LIN {X 0,Y 129.173,Z 379.611,A -85,B 0,C 180,E1 -25427.278,E2 -25427.278} C_VEL
LIN {X 0,Y 127.042,Z 350.906,A -85,B 0,C 180,E1 -25430.039,E2 -25430.039} C_VEL
LIN {X 0,Y 126.624,Z 346.55,A -85,B 0,C 180,E1 -25430.476,E2 -25430.476} C_VEL
LIN {X 0,Y 125.446,Z 341.472,A -85,B 0,C 180,E1 -25431.146,E2 -25431.146} C_VEL
LIN {X 0,Y 123.586,Z 332.403,A -85,B 0,C 180,E1 -25437.298,E2 -25437.298} C_VEL
LIN {X 0,Y 122.03,Z 325.286,A -85,B 0,C 180,E1 -25442.561,E2 -25442.561} C_VEL
LIN {X 0,Y 121.994,Z 325.288,A -85,B 0,C 180,E1 -25449.773,E2 -25449.773} C_VEL
LIN {X 0,Y 122.194,Z 325.256,A -85,B 0,C 180,E1 -25456.694,E2 -25456.694} C_VEL
LIN {X 0,Y 122.396,Z 325.238,A -85,B 0,C 180,E1 -25460.075,E2 -25460.075} C_VEL
LIN {X 0,Y 122.56,Z 325.214,A -85,B 0,C 180,E1 -25466.706,E2 -25466.706} C_VEL
LIN {X 0,Y 123.024,Z 325.16,A -85,B 0,C 180,E1 -25469.993,E2 -25469.993} C_VEL
LIN {X 0,Y 122.41,Z 325.236,A -85,B 0,C 180,E1 -25476.586,E2 -25476.586} C_VEL
LIN {X 0,Y 122.397,Z 325.238,A -85,B 0,C 180,E1 -25479.911,E2 -25479.911} C_VEL
LIN {X 0,Y 122.188,Z 325.258,A -85,B 0,C 180,E1 -25483.293,E2 -25483.293} C_VEL
LIN {X 0,Y 121.987,Z 325.286,A -85,B 0,C 180,E1 -25490.214,E2 -25490.214} C_VEL
LIN {X 0,Y 121.947,Z 325.292,A -85,B 0,C 180,E1 -25493.782,E2 -25493.782} C_VEL
LIN {X 0,Y 121.919,Z 325.29,A -85,B 0,C 180,E1 -25500.151,E2 -25500.151} C_VEL
LIN {X 0,Y 121.87,Z 325.303,A -85,B 0,C 180,E1 -25506.159,E2 -25506.159} C_VEL
LIN {X 0,Y 121.85,Z 325.303,A -85,B 0,C 180,E1 -25511.423,E2 -25511.423} C_VEL
LIN {X 0,Y 121.846,Z 325.3,A -85,B 0,C 180,E1 -25518.559,E2 -25518.559} C_VEL
LIN {X 0,Y 121.889,Z 325.3,A -85,B 0,C 180,E1 -25524.787,E2 -25524.787} C_VEL
LIN {X 0,Y 121.907,Z 325.298,A -85,B 0,C 180,E1 -25529.832,E2 -25529.832} C_VEL
LIN {X 0,Y 121.931,Z 325.289,A -85,B 0,C 180,E1 -25536.203,E2 -25536.203} C_VEL
LIN {X 0,Y 121.964,Z 325.293,A -85,B 0,C 180,E1 -25539.771,E2 -25539.771} C_VEL
LIN {X 0,Y 122.161,Z 325.265,A -85,B 0,C 180,E1 -25546.694,E2 -25546.694} C_VEL
LIN {X 0,Y 122.367,Z 325.243,A -85,B 0,C 180,E1 -25550.077,E2 -25550.077} C_VEL
LIN {X 0,Y 122.562,Z 325.217,A -85,B 0,C 180,E1 -25556.711,E2 -25556.711} C_VEL
LIN {X 0,Y 123.006,Z 325.161,A -85,B 0,C 180,E1 -25559.998,E2 -25559.998} C_VEL
LIN {X 0,Y 122.387,Z 325.239,A -85,B 0,C 180,E1 -25566.593,E2 -25566.593} C_VEL
LIN {X 0,Y 122.367,Z 325.238,A -85,B 0,C 180,E1 -25569.92,E2 -25569.92} C_VEL
LIN {X 0,Y 122.055,Z 325.28,A -85,B 0,C 180,E1 -25576.731,E2 -25576.731} C_VEL
LIN {X 0,Y 122.002,Z 325.286,A -85,B 0,C 180,E1 -25582.856,E2 -25582.856} C_VEL
LIN {X 0,Y 121.914,Z 325.296,A -85,B 0,C 180,E1 -25587.461,E2 -25587.461} C_VEL
LIN {X 0,Y 121.874,Z 325.301,A -85,B 0,C 180,E1 -25591.263,E2 -25591.263} C_VEL
LIN {X 0,Y 121.856,Z 325.304,A -85,B 0,C 180,E1 -25596.172,E2 -25596.172} C_VEL
LIN {X 0,Y 121.899,Z 325.302,A -85,B 0,C 180,E1 -25603.44,E2 -25603.44} C_VEL
LIN {X 0,Y 123.968,Z 334.356,A -85,B 0,C 180,E1 -25609.71,E2 -25609.71} C_VEL
LIN {X 0,Y 125.965,Z 343.489,A -85,B 0,C 180,E1 -25615.496,E2 -25615.496} C_VEL
LIN {X 0,Y 129.129,Z 356.128,A -85,B 0,C 180,E1 -25616.87,E2 -25616.87} C_VEL
LIN {X 0,Y 130.258,Z 379.545,A -85,B 0,C 180,E1 -25618.925,E2 -25618.925} C_VEL
LIN {X 0,Y 130.546,Z 387.282,A -85,B 0,C 180,E1 -25619.591,E2 -25619.591} C_VEL
LIN {X 0,Y 127.713,Z 439.812,A -85,B 0,C 180,E1 -25624.001,E2 -25624.001} C_VEL
LIN {X 0,Y 127.078,Z 449.021,A -85,B 0,C 180,E1 -25625.068,E2 -25625.068} C_VEL
LIN {X 0,Y 126.116,Z 458.949,A -85,B 0,C 180,E1 -25626.616,E2 -25626.616} C_VEL
LIN {X 0,Y 125.046,Z 468.69,A -85,B 0,C 180,E1 -25628.582,E2 -25628.582} C_VEL
LIN {X 0,Y 124.012,Z 478.18,A -85,B 0,C 180,E1 -25630.991,E2 -25630.991} C_VEL
LIN {X 0,Y 122.965,Z 487.212,A -85,B 0,C 180,E1 -25633.83,E2 -25633.83} C_VEL
LIN {X 0,Y 122.171,Z 494.773,A -85,B 0,C 180,E1 -25636.705,E2 -25636.705} C_VEL
LIN {X 0,Y 121.656,Z 502.106,A -85,B 0,C 180,E1 -25640.028,E2 -25640.028} C_VEL
LIN {X 0,Y 121.435,Z 508.305,A -85,B 0,C 180,E1 -25643.361,E2 -25643.361} C_VEL
LIN {X 0,Y 121.501,Z 513.6,A -85,B 0,C 180,E1 -25646.691,E2 -25646.691} C_VEL
LIN {X 0,Y 121.483,Z 517.958,A -85,B 0,C 180,E1 -25650.007,E2 -25650.007} C_VEL
LIN {X 0,Y 121.523,Z 519.76,A -85,B 0,C 180,E1 -25651.664,E2 -25651.664} C_VEL
LIN {X 0,Y 120.888,Z 524.223,A -85,B 0,C 180,E1 -25656.683,E2 -25656.683} C_VEL
LIN {X 0,Y 120.757,Z 526.661,A -85,B 0,C 180,E1 -25660.061,E2 -25660.061} C_VEL
LIN {X 0,Y 122.013,Z 530.169,A -85,B 0,C 180,E1 -25666.744,E2 -25666.744} C_VEL
LIN {X 0,Y 125.047,Z 532.186,A -85,B 0,C 180,E1 -25673.172,E2 -25673.172} C_VEL
LIN {X 0,Y 127.347,Z 532.797,A -85,B 0,C 180,E1 -25676.204,E2 -25676.204} C_VEL
LIN {X 0,Y 132.935,Z 532.734,A -85,B 0,C 180,E1 -25681.92,E2 -25681.92} C_VEL
LIN {X 0,Y 140.05,Z 531.292,A -85,B 0,C 180,E1 -25687.029,E2 -25687.029} C_VEL
LIN {X 0,Y 144.169,Z 530.134,A -85,B 0,C 180,E1 -25689.328,E2 -25689.328} C_VEL
LIN {X 0,Y 153.238,Z 526.471,A -85,B 0,C 180,E1 -25693.47,E2 -25693.47} C_VEL
LIN {X 0,Y 160.656,Z 522.679,A -85,B 0,C 180,E1 -25696.205,E2 -25696.205} C_VEL
LIN {X 0,Y 168.584,Z 517.857,A -85,B 0,C 180,E1 -25698.625,E2 -25698.625} C_VEL
LIN {X 0,Y 176.893,Z 511.872,A -85,B 0,C 180,E1 -25700.782,E2 -25700.782} C_VEL
LIN {X 0,Y 182.966,Z 506.877,A -85,B 0,C 180,E1 -25702.125,E2 -25702.125} C_VEL
LIN {X 0,Y 186.444,Z 503.636,A -85,B 0,C 180,E1 -25702.865,E2 -25702.865} C_VEL
LIN {X 0,Y 187.553,Z 502.508,A -85,B 0,C 180,E1 -25703.38,E2 -25703.38} C_VEL
LIN {X 0,Y 187.967,Z 501.842,A -85,B 0,C 180,E1 -25704.343,E2 -25704.343} C_VEL
LIN {X 0,Y 187.307,Z 502.027,A -85,B 0,C 180,E1 -25705.711,E2 -25705.711} C_VEL
LIN {X 0,Y 185.694,Z 503.089,A -85,B 0,C 180,E1 -25707.077,E2 -25707.077} C_VEL
LIN {X 0,Y 183.227,Z 504.981,A -85,B 0,C 180,E1 -25708.567,E2 -25708.567} C_VEL
LIN {X 0,Y 179.601,Z 507.677,A -85,B 0,C 180,E1 -25710.16,E2 -25710.16} C_VEL
LIN {X 0,Y 176.658,Z 509.754,A -85,B 0,C 180,E1 -25711.01,E2 -25711.01} C_VEL
LIN {X 0,Y 169.265,Z 514.461,A -85,B 0,C 180,E1 -25712.825,E2 -25712.825} C_VEL
LIN {X 0,Y 163.188,Z 517.73,A -85,B 0,C 180,E1 -25714.491,E2 -25714.491} C_VEL
LIN {X 0,Y 154.625,Z 521.426,A -85,B 0,C 180,E1 -25717.275,E2 -25717.275} C_VEL
LIN {X 0,Y 150.902,Z 522.795,A -85,B 0,C 180,E1 -25718.665,E2 -25718.665} C_VEL
LIN {X 0,Y 141.546,Z 525.001,A -85,B 0,C 180,E1 -25722.669,E2 -25722.669} C_VEL
LIN {X 0,Y 136.899,Z 525.619,A -85,B 0,C 180,E1 -25725.128,E2 -25725.128} C_VEL
LIN {X 0,Y 132.534,Z 525.668,A -85,B 0,C 180,E1 -25727.755,E2 -25727.755} C_VEL
LIN {X 0,Y 125.02,Z 524.446,A -85,B 0,C 180,E1 -25733.546,E2 -25733.546} C_VEL
LIN {X 0,Y 121.894,Z 523.17,A -85,B 0,C 180,E1 -25736.696,E2 -25736.696} C_VEL
LIN {X 0,Y 118.039,Z 520.332,A -85,B 0,C 180,E1 -25741.708,E2 -25741.708} C_VEL
LIN {X 0,Y 115.253,Z 516.339,A -85,B 0,C 180,E1 -25747.007,E2 -25747.007} C_VEL
LIN {X 0,Y 113.524,Z 511.07,A -85,B 0,C 180,E1 -25752.516,E2 -25752.516} C_VEL
LIN {X 0,Y 112.939,Z 505.58,A -85,B 0,C 180,E1 -25757.195,E2 -25757.195} C_VEL
LIN {X 0,Y 113.016,Z 498.844,A -85,B 0,C 180,E1 -25761.91,E2 -25761.91} C_VEL
LIN {X 0,Y 113.405,Z 492.3,A -85,B 0,C 180,E1 -25765.712,E2 -25765.712} C_VEL
LIN {X 0,Y 114.052,Z 484.365,A -85,B 0,C 180,E1 -25769.538,E2 -25769.538} C_VEL
LIN {X 0,Y 114.935,Z 475.882,A -85,B 0,C 180,E1 -25772.895,E2 -25772.895} C_VEL
LIN {X 0,Y 115.837,Z 467.102,A -85,B 0,C 180,E1 -25775.732,E2 -25775.732} C_VEL
LIN {X 0,Y 117.087,Z 455.66,A -85,B 0,C 180,E1 -25778.707,E2 -25778.707} C_VEL
LIN {X 0,Y 118.276,Z 443.044,A -85,B 0,C 180,E1 -25781.1,E2 -25781.1} C_VEL
LIN {X 0,Y 118.993,Z 433.1,A -85,B 0,C 180,E1 -25782.497,E2 -25782.497} C_VEL
LIN {X 0,Y 121.054,Z 399.59,A -85,B 0,C 180,E1 -25785.835,E2 -25785.835} C_VEL
LIN {X 0,Y 122.178,Z 380.662,A -85,B 0,C 180,E1 -25787.614,E2 -25787.614} C_VEL
LIN {X 0,Y 120.099,Z 351.697,A -85,B 0,C 180,E1 -25790.566,E2 -25790.566} C_VEL
LIN {X 0,Y 119.618,Z 347.583,A -85,B 0,C 180,E1 -25791.012,E2 -25791.012} C_VEL
LIN {X 0,Y 118.244,Z 341.693,A -85,B 0,C 180,E1 -25791.746,E2 -25791.746} C_VEL
LIN {X 0,Y 116.561,Z 333.547,A -85,B 0,C 180,E1 -25797.581,E2 -25797.581} C_VEL
LIN {X 0,Y 114.949,Z 326.167,A -85,B 0,C 180,E1 -25803.315,E2 -25803.315} C_VEL
LIN {X 0,Y 114.928,Z 326.171,A -85,B 0,C 180,E1 -25808.47,E2 -25808.47} C_VEL
LIN {X 0,Y 114.972,Z 326.163,A -85,B 0,C 180,E1 -25812.198,E2 -25812.198} C_VEL
LIN {X 0,Y 115.311,Z 326.122,A -85,B 0,C 180,E1 -25819.458,E2 -25819.458} C_VEL
LIN {X 0,Y 115.487,Z 326.095,A -85,B 0,C 180,E1 -25826.504,E2 -25826.504} C_VEL
LIN {X 0,Y 115.975,Z 326.038,A -85,B 0,C 180,E1 -25829.993,E2 -25829.993} C_VEL
LIN {X 0,Y 115.352,Z 326.115,A -85,B 0,C 180,E1 -25836.991,E2 -25836.991} C_VEL
LIN {X 0,Y 115.205,Z 326.127,A -85,B 0,C 180,E1 -25842.552,E2 -25842.552} C_VEL
LIN {X 0,Y 114.966,Z 326.163,A -85,B 0,C 180,E1 -25847.788,E2 -25847.788} C_VEL
LIN {X 0,Y 114.91,Z 326.168,A -85,B 0,C 180,E1 -25853.445,E2 -25853.445} C_VEL
LIN {X 0,Y 114.847,Z 326.171,A -85,B 0,C 180,E1 -25861.046,E2 -25861.046} C_VEL
LIN {X 0,Y 114.763,Z 326.186,A -85,B 0,C 180,E1 -25867.749,E2 -25867.749} C_VEL
LIN {X 0,Y 114.764,Z 326.189,A -85,B 0,C 180,E1 -25872.702,E2 -25872.702} C_VEL
LIN {X 0,Y 114.77,Z 326.183,A -85,B 0,C 180,E1 -25877.652,E2 -25877.652} C_VEL
LIN {X 0,Y 114.765,Z 326.19,A -85,B 0,C 180,E1 -25882.739,E2 -25882.739} C_VEL
LIN {X 0,Y 114.836,Z 326.176,A -85,B 0,C 180,E1 -25888.936,E2 -25888.936} C_VEL
LIN {X 0,Y 114.894,Z 326.165,A -85,B 0,C 180,E1 -25896.538,E2 -25896.538} C_VEL
LIN {X 0,Y 114.939,Z 326.166,A -85,B 0,C 180,E1 -25902.196,E2 -25902.196} C_VEL
LIN {X 0,Y 115.281,Z 326.124,A -85,B 0,C 180,E1 -25909.46,E2 -25909.46} C_VEL
LIN {X 0,Y 115.486,Z 326.097,A -85,B 0,C 180,E1 -25916.509,E2 -25916.509} C_VEL
LIN {X 0,Y 115.958,Z 326.039,A -85,B 0,C 180,E1 -25919.998,E2 -25919.998} C_VEL
LIN {X 0,Y 115.328,Z 326.119,A -85,B 0,C 180,E1 -25926.999,E2 -25926.999} C_VEL
LIN {X 0,Y 115.179,Z 326.132,A -85,B 0,C 180,E1 -25932.56,E2 -25932.56} C_VEL
LIN {X 0,Y 114.963,Z 326.164,A -85,B 0,C 180,E1 -25937.796,E2 -25937.796} C_VEL
LIN {X 0,Y 114.92,Z 326.168,A -85,B 0,C 180,E1 -25943.492,E2 -25943.492} C_VEL
LIN {X 0,Y 114.831,Z 326.177,A -85,B 0,C 180,E1 -25951.059,E2 -25951.059} C_VEL
LIN {X 0,Y 114.751,Z 326.193,A -85,B 0,C 180,E1 -25957.765,E2 -25957.765} C_VEL
LIN {X 0,Y 114.842,Z 326.253,A -85,B 0,C 180,E1 -25962.763,E2 -25962.763} C_VEL
LIN {X 0,Y 116.972,Z 335.554,A -85,B 0,C 180,E1 -25969.512,E2 -25969.512} C_VEL
LIN {X 0,Y 118.738,Z 343.603,A -85,B 0,C 180,E1 -25974.831,E2 -25974.831} C_VEL
LIN {X 0,Y 122.146,Z 357.637,A -85,B 0,C 180,E1 -25976.43,E2 -25976.43} C_VEL
LIN {X 0,Y 123.485,Z 387.391,A -85,B 0,C 180,E1 -25979.199,E2 -25979.199} C_VEL
LIN {X 0,Y 120.627,Z 439.492,A -85,B 0,C 180,E1 -25983.868,E2 -25983.868} C_VEL
LIN {X 0,Y 119.905,Z 449.334,A -85,B 0,C 180,E1 -25985.095,E2 -25985.095} C_VEL
LIN {X 0,Y 118.97,Z 459.137,A -85,B 0,C 180,E1 -25986.741,E2 -25986.741} C_VEL
LIN {X 0,Y 117.831,Z 469.633,A -85,B 0,C 180,E1 -25989.04,E2 -25989.04} C_VEL
LIN {X 0,Y 116.793,Z 478.856,A -85,B 0,C 180,E1 -25991.593,E2 -25991.593} C_VEL
LIN {X 0,Y 115.81,Z 487.711,A -85,B 0,C 180,E1 -25994.612,E2 -25994.612} C_VEL
LIN {X 0,Y 115.05,Z 496.154,A -85,B 0,C 180,E1 -25998.123,E2 -25998.123} C_VEL
LIN {X 0,Y 114.617,Z 504.09,A -85,B 0,C 180,E1 -26002.176,E2 -26002.176} C_VEL
LIN {X 0,Y 114.643,Z 512.313,A -85,B 0,C 180,E1 -26007.372,E2 -26007.372} C_VEL
LIN {X 0,Y 114.675,Z 517.684,A -85,B 0,C 180,E1 -26011.763,E2 -26011.763} C_VEL
LIN {X 0,Y 114.045,Z 522.48,A -85,B 0,C 180,E1 -26017.086,E2 -26017.086} C_VEL
LIN {X 0,Y 114.402,Z 527.08,A -85,B 0,C 180,E1 -26024.231,E2 -26024.231} C_VEL
LIN {X 0,Y 115.32,Z 528.858,A -85,B 0,C 180,E1 -26027.747,E2 -26027.747} C_VEL
LIN {X 0,Y 118.58,Z 531.297,A -85,B 0,C 180,E1 -26034.516,E2 -26034.516} C_VEL
LIN {X 0,Y 123.784,Z 532.278,A -85,B 0,C 180,E1 -26040.734,E2 -26040.734} C_VEL
LIN {X 0,Y 128.713,Z 532.194,A -85,B 0,C 180,E1 -26045.015,E2 -26045.015} C_VEL
LIN {X 0,Y 134.453,Z 531.346,A -85,B 0,C 180,E1 -26048.851,E2 -26048.851} C_VEL
LIN {X 0,Y 143.291,Z 528.883,A -85,B 0,C 180,E1 -26053.368,E2 -26053.368} C_VEL
LIN {X 0,Y 150.718,Z 526.081,A -85,B 0,C 180,E1 -26056.285,E2 -26056.285} C_VEL
LIN {X 0,Y 158.553,Z 522.398,A -85,B 0,C 180,E1 -26058.899,E2 -26058.899} C_VEL
LIN {X 0,Y 166.866,Z 517.646,A -85,B 0,C 180,E1 -26061.186,E2 -26061.186} C_VEL
LIN {X 0,Y 175.517,Z 511.729,A -85,B 0,C 180,E1 -26063.21,E2 -26063.21} C_VEL
LIN {X 0,Y 183.776,Z 505.127,A -85,B 0,C 180,E1 -26064.843,E2 -26064.843} C_VEL
LIN {X 0,Y 190.678,Z 498.721,A -85,B 0,C 180,E1 -26066.026,E2 -26066.026} C_VEL
LIN {X 0,Y 195.373,Z 493.88,A -85,B 0,C 180,E1 -26066.764,E2 -26066.764} C_VEL
LIN {X 0,Y 195.249,Z 493.91,A -85,B 0,C 180,E1 -26067.323,E2 -26067.323} C_VEL
LIN {X 0,Y 186.903,Z 501.833,A -85,B 0,C 180,E1 -26068.868,E2 -26068.868} C_VEL
LIN {X 0,Y 179.375,Z 507.837,A -85,B 0,C 180,E1 -26070.407,E2 -26070.407} C_VEL
LIN {X 0,Y 176.658,Z 509.754,A -85,B 0,C 180,E1 -26071.01,E2 -26071.01} C_VEL
LIN {X 0,Y 172.145,Z 512.757,A -85,B 0,C 180,E1 -26071.818,E2 -26071.818} C_VEL
LIN {X 0,Y 163.776,Z 517.343,A -85,B 0,C 180,E1 -26072.782,E2 -26072.782} C_VEL
LIN {X 0,Y 155.281,Z 521.101,A -85,B 0,C 180,E1 -26073.952,E2 -26073.952} C_VEL
LIN {X 0,Y 150.639,Z 522.727,A -85,B 0,C 180,E1 -26075.114,E2 -26075.114} C_VEL
LIN {X 0,Y 144.865,Z 524.313,A -85,B 0,C 180,E1 -26077.164,E2 -26077.164} C_VEL
LIN {X 0,Y 139.439,Z 525.432,A -85,B 0,C 180,E1 -26079.342,E2 -26079.342} C_VEL
LIN {X 0,Y 132.579,Z 526.179,A -85,B 0,C 180,E1 -26082.591,E2 -26082.591} C_VEL
LIN {X 0,Y 125.145,Z 525.88,A -85,B 0,C 180,E1 -26087.02,E2 -26087.02} C_VEL
LIN {X 0,Y 121.121,Z 525.186,A -85,B 0,C 180,E1 -26089.977,E2 -26089.977} C_VEL
LIN {X 0,Y 117.53,Z 523.906,A -85,B 0,C 180,E1 -26093.133,E2 -26093.133} C_VEL
LIN {X 0,Y 111.73,Z 520.067,A -85,B 0,C 180,E1 -26100.002,E2 -26100.002} C_VEL
LIN {X 0,Y 108.67,Z 515.851,A -85,B 0,C 180,E1 -26105.569,E2 -26105.569} C_VEL
LIN {X 0,Y 107.078,Z 511.736,A -85,B 0,C 180,E1 -26110.085,E2 -26110.085} C_VEL
LIN {X 0,Y 106.121,Z 505.974,A -85,B 0,C 180,E1 -26115.363,E2 -26115.363} C_VEL
LIN {X 0,Y 105.959,Z 500.857,A -85,B 0,C 180,E1 -26119.37,E2 -26119.37} C_VEL
LIN {X 0,Y 106.315,Z 492.91,A -85,B 0,C 180,E1 -26124.406,E2 -26124.406} C_VEL
LIN {X 0,Y 106.992,Z 483.988,A -85,B 0,C 180,E1 -26128.978,E2 -26128.978} C_VEL
LIN {X 0,Y 107.971,Z 474.349,A -85,B 0,C 180,E1 -26132.979,E2 -26132.979} C_VEL
LIN {X 0,Y 109.103,Z 463.38,A -85,B 0,C 180,E1 -26136.576,E2 -26136.576} C_VEL
LIN {X 0,Y 110.273,Z 452.568,A -85,B 0,C 180,E1 -26139.3,E2 -26139.3} C_VEL
LIN {X 0,Y 111.336,Z 441.435,A -85,B 0,C 180,E1 -26141.426,E2 -26141.426} C_VEL
LIN {X 0,Y 112.092,Z 429.813,A -85,B 0,C 180,E1 -26143.045,E2 -26143.045} C_VEL
LIN {X 0,Y 115.18,Z 381.489,A -85,B 0,C 180,E1 -26147.979,E2 -26147.979} C_VEL
LIN {X 0,Y 113.117,Z 351.719,A -85,B 0,C 180,E1 -26151.205,E2 -26151.205} C_VEL
LIN {X 0,Y 111.937,Z 345.593,A -85,B 0,C 180,E1 -26151.965,E2 -26151.965} C_VEL
LIN {X 0,Y 111.009,Z 341.617,A -85,B 0,C 180,E1 -26152.595,E2 -26152.595} C_VEL
LIN {X 0,Y 109.251,Z 333.22,A -85,B 0,C 180,E1 -26159.022,E2 -26159.022} C_VEL
LIN {X 0,Y 107.849,Z 327.053,A -85,B 0,C 180,E1 -26164.14,E2 -26164.14} C_VEL
LIN {X 0,Y 107.864,Z 327.049,A -85,B 0,C 180,E1 -26170.981,E2 -26170.981} C_VEL
LIN {X 0,Y 108.211,Z 327.003,A -85,B 0,C 180,E1 -26178.758,E2 -26178.758} C_VEL
LIN {X 0,Y 108.291,Z 326.994,A -85,B 0,C 180,E1 -26182.535,E2 -26182.535} C_VEL
LIN {X 0,Y 108.901,Z 326.92,A -85,B 0,C 180,E1 -26189.993,E2 -26189.993} C_VEL
LIN {X 0,Y 108.292,Z 326.995,A -85,B 0,C 180,E1 -26197.45,E2 -26197.45} C_VEL
LIN {X 0,Y 108.139,Z 327.007,A -85,B 0,C 180,E1 -26202.866,E2 -26202.866} C_VEL
LIN {X 0,Y 107.862,Z 327.047,A -85,B 0,C 180,E1 -26209.003,E2 -26209.003} C_VEL
LIN {X 0,Y 107.825,Z 327.051,A -85,B 0,C 180,E1 -26214.14,E2 -26214.14} C_VEL
LIN {X 0,Y 107.77,Z 327.056,A -85,B 0,C 180,E1 -26222.027,E2 -26222.027} C_VEL
LIN {X 0,Y 107.671,Z 327.066,A -85,B 0,C 180,E1 -26228.435,E2 -26228.435} C_VEL
LIN {X 0,Y 107.654,Z 327.074,A -85,B 0,C 180,E1 -26235.882,E2 -26235.882} C_VEL
LIN {X 0,Y 107.665,Z 327.072,A -85,B 0,C 180,E1 -26241.546,E2 -26241.546} C_VEL
LIN {X 0,Y 107.772,Z 327.054,A -85,B 0,C 180,E1 -26248.552,E2 -26248.552} C_VEL
LIN {X 0,Y 107.858,Z 327.042,A -85,B 0,C 180,E1 -26256.984,E2 -26256.984} C_VEL
LIN {X 0,Y 107.943,Z 327.03,A -85,B 0,C 180,E1 -26264.902,E2 -26264.902} C_VEL
LIN {X 0,Y 108.199,Z 327.007,A -85,B 0,C 180,E1 -26268.761,E2 -26268.761} C_VEL
LIN {X 0,Y 108.41,Z 326.978,A -85,B 0,C 180,E1 -26276.281,E2 -26276.281} C_VEL
LIN {X 0,Y 108.884,Z 326.92,A -85,B 0,C 180,E1 -26279.998,E2 -26279.998} C_VEL
LIN {X 0,Y 108.267,Z 326.999,A -85,B 0,C 180,E1 -26287.458,E2 -26287.458} C_VEL
LIN {X 0,Y 108.113,Z 327.012,A -85,B 0,C 180,E1 -26292.874,E2 -26292.874} C_VEL
LIN {X 0,Y 107.862,Z 327.045,A -85,B 0,C 180,E1 -26299.011,E2 -26299.011} C_VEL
LIN {X 0,Y 107.83,Z 327.053,A -85,B 0,C 180,E1 -26304.182,E2 -26304.182} C_VEL
LIN {X 0,Y 107.754,Z 327.06,A -85,B 0,C 180,E1 -26312.04,E2 -26312.04} C_VEL
LIN {X 0,Y 107.671,Z 327.075,A -85,B 0,C 180,E1 -26318.458,E2 -26318.458} C_VEL
LIN {X 0,Y 107.75,Z 327.164,A -85,B 0,C 180,E1 -26321.89,E2 -26321.89} C_VEL
LIN {X 0,Y 109.811,Z 336.039,A -85,B 0,C 180,E1 -26328.762,E2 -26328.762} C_VEL
LIN {X 0,Y 111.475,Z 343.518,A -85,B 0,C 180,E1 -26334.067,E2 -26334.067} C_VEL
LIN {X 0,Y 115.169,Z 358.51,A -85,B 0,C 180,E1 -26335.917,E2 -26335.917} C_VEL
LIN {X 0,Y 116.429,Z 387.557,A -85,B 0,C 180,E1 -26338.79,E2 -26338.79} C_VEL
LIN {X 0,Y 113.507,Z 440.129,A -85,B 0,C 180,E1 -26343.833,E2 -26343.833} C_VEL
LIN {X 0,Y 112.775,Z 449.689,A -85,B 0,C 180,E1 -26345.135,E2 -26345.135} C_VEL
LIN {X 0,Y 111.816,Z 459.289,A -85,B 0,C 180,E1 -26346.88,E2 -26346.88} C_VEL
LIN {X 0,Y 110.788,Z 468.754,A -85,B 0,C 180,E1 -26349.104,E2 -26349.104} C_VEL
LIN {X 0,Y 109.939,Z 476.61,A -85,B 0,C 180,E1 -26351.369,E2 -26351.369} C_VEL
LIN {X 0,Y 108.944,Z 485.692,A -85,B 0,C 180,E1 -26354.577,E2 -26354.577} C_VEL
LIN {X 0,Y 108.164,Z 494.366,A -85,B 0,C 180,E1 -26358.338,E2 -26358.338} C_VEL
LIN {X 0,Y 107.764,Z 502.271,A -85,B 0,C 180,E1 -26362.514,E2 -26362.514} C_VEL
LIN {X 0,Y 107.771,Z 508.216,A -85,B 0,C 180,E1 -26366.269,E2 -26366.269} C_VEL
LIN {X 0,Y 107.85,Z 513.205,A -85,B 0,C 180,E1 -26370.008,E2 -26370.008} C_VEL
LIN {X 0,Y 107.724,Z 517.319,A -85,B 0,C 180,E1 -26373.748,E2 -26373.748} C_VEL
LIN {X 0,Y 107.173,Z 522.537,A -85,B 0,C 180,E1 -26380.389,E2 -26380.389} C_VEL
LIN {X 0,Y 107.702,Z 525.517,A -85,B 0,C 180,E1 -26385.137,E2 -26385.137} C_VEL
LIN {X 0,Y 110.167,Z 528.969,A -85,B 0,C 180,E1 -26392.511,E2 -26392.511} C_VEL
LIN {X 0,Y 114.837,Z 531.01,A -85,B 0,C 180,E1 -26399.319,E2 -26399.319} C_VEL
LIN {X 0,Y 117.737,Z 531.604,A -85,B 0,C 180,E1 -26402.5,E2 -26402.5} C_VEL
LIN {X 0,Y 124.879,Z 531.67,A -85,B 0,C 180,E1 -26408.251,E2 -26408.251} C_VEL
LIN {X 0,Y 133.491,Z 530.335,A -85,B 0,C 180,E1 -26413.193,E2 -26413.193} C_VEL
LIN {X 0,Y 138.224,Z 529.224,A -85,B 0,C 180,E1 -26415.387,E2 -26415.387} C_VEL
LIN {X 0,Y 148.542,Z 525.79,A -85,B 0,C 180,E1 -26419.203,E2 -26419.203} C_VEL
LIN {X 0,Y 156.816,Z 522.15,A -85,B 0,C 180,E1 -26421.657,E2 -26421.657} C_VEL
LIN {X 0,Y 165.501,Z 517.524,A -85,B 0,C 180,E1 -26423.788,E2 -26423.788} C_VEL
LIN {X 0,Y 174.882,Z 511.444,A -85,B 0,C 180,E1 -26425.716,E2 -26425.716} C_VEL
LIN {X 0,Y 180.57,Z 507.239,A -85,B 0,C 180,E1 -26426.75,E2 -26426.75} C_VEL
LIN {X 0,Y 182.251,Z 505.801,A -85,B 0,C 180,E1 -26427.326,E2 -26427.326} C_VEL
LIN {X 0,Y 171.246,Z 513.262,A -85,B 0,C 180,E1 -26429.524,E2 -26429.524} C_VEL
LIN {X 0,Y 162.55,Z 517.891,A -85,B 0,C 180,E1 -26431.603,E2 -26431.603} C_VEL
LIN {X 0,Y 156.426,Z 520.653,A -85,B 0,C 180,E1 -26433.304,E2 -26433.304} C_VEL
LIN {X 0,Y 150.639,Z 522.727,A -85,B 0,C 180,E1 -26435.114,E2 -26435.114} C_VEL
LIN {X 0,Y 147.349,Z 523.782,A -85,B 0,C 180,E1 -26435.896,E2 -26435.896} C_VEL
LIN {X 0,Y 141.039,Z 525.33,A -85,B 0,C 180,E1 -26436.675,E2 -26436.675} C_VEL
LIN {X 0,Y 134.731,Z 526.369,A -85,B 0,C 180,E1 -26437.564,E2 -26437.564} C_VEL
LIN {X 0,Y 131.496,Z 526.626,A -85,B 0,C 180,E1 -26438.551,E2 -26438.551} C_VEL
LIN {X 0,Y 122.271,Z 526.506,A -85,B 0,C 180,E1 -26443.3,E2 -26443.3} C_VEL
LIN {X 0,Y 117.777,Z 525.859,A -85,B 0,C 180,E1 -26446.193,E2 -26446.193} C_VEL
LIN {X 0,Y 110.081,Z 523.023,A -85,B 0,C 180,E1 -26452.666,E2 -26452.666} C_VEL
LIN {X 0,Y 105.478,Z 519.659,A -85,B 0,C 180,E1 -26458.164,E2 -26458.164} C_VEL
LIN {X 0,Y 102.184,Z 515.306,A -85,B 0,C 180,E1 -26463.946,E2 -26463.946} C_VEL
LIN {X 0,Y 100.176,Z 510.191,A -85,B 0,C 180,E1 -26469.576,E2 -26469.576} C_VEL
LIN {X 0,Y 99.206,Z 503.818,A -85,B 0,C 180,E1 -26475.408,E2 -26475.408} C_VEL
LIN {X 0,Y 99.173,Z 495.711,A -85,B 0,C 180,E1 -26481.499,E2 -26481.499} C_VEL
LIN {X 0,Y 99.69,Z 486.859,A -85,B 0,C 180,E1 -26486.71,E2 -26486.71} C_VEL
LIN {X 0,Y 100.37,Z 479.044,A -85,B 0,C 180,E1 -26490.453,E2 -26490.453} C_VEL
LIN {X 0,Y 101.191,Z 470.74,A -85,B 0,C 180,E1 -26493.756,E2 -26493.756} C_VEL
LIN {X 0,Y 102.221,Z 460.73,A -85,B 0,C 180,E1 -26496.986,E2 -26496.986} C_VEL
LIN {X 0,Y 103.224,Z 451.597,A -85,B 0,C 180,E1 -26499.352,E2 -26499.352} C_VEL
LIN {X 0,Y 104.235,Z 441.264,A -85,B 0,C 180,E1 -26501.446,E2 -26501.446} C_VEL
LIN {X 0,Y 105.072,Z 428.849,A -85,B 0,C 180,E1 -26503.283,E2 -26503.283} C_VEL
LIN {X 0,Y 108.147,Z 381.797,A -85,B 0,C 180,E1 -26508.447,E2 -26508.447} C_VEL
LIN {X 0,Y 105.969,Z 350.894,A -85,B 0,C 180,E1 -26512.003,E2 -26512.003} C_VEL
LIN {X 0,Y 103.793,Z 341.7,A -85,B 0,C 180,E1 -26513.359,E2 -26513.359} C_VEL
LIN {X 0,Y 102.046,Z 333.567,A -85,B 0,C 180,E1 -26520.04,E2 -26520.04} C_VEL
LIN {X 0,Y 100.808,Z 327.929,A -85,B 0,C 180,E1 -26525.007,E2 -26525.007} C_VEL
LIN {X 0,Y 100.777,Z 327.932,A -85,B 0,C 180,E1 -26529.586,E2 -26529.586} C_VEL
LIN {X 0,Y 101.121,Z 327.885,A -85,B 0,C 180,E1 -26537.958,E2 -26537.958} C_VEL
LIN {X 0,Y 101.225,Z 327.874,A -85,B 0,C 180,E1 -26542.011,E2 -26542.011} C_VEL
LIN {X 0,Y 101.828,Z 327.801,A -85,B 0,C 180,E1 -26549.992,E2 -26549.992} C_VEL
LIN {X 0,Y 101.229,Z 327.876,A -85,B 0,C 180,E1 -26557.973,E2 -26557.973} C_VEL
LIN {X 0,Y 101.051,Z 327.89,A -85,B 0,C 180,E1 -26563.164,E2 -26563.164} C_VEL
LIN {X 0,Y 100.779,Z 327.926,A -85,B 0,C 180,E1 -26570.396,E2 -26570.396} C_VEL
LIN {X 0,Y 100.73,Z 327.936,A -85,B 0,C 180,E1 -26574.898,E2 -26574.898} C_VEL
LIN {X 0,Y 100.679,Z 327.941,A -85,B 0,C 180,E1 -26583.101,E2 -26583.101} C_VEL
LIN {X 0,Y 100.622,Z 327.943,A -85,B 0,C 180,E1 -26589.795,E2 -26589.795} C_VEL
LIN {X 0,Y 100.625,Z 327.949,A -85,B 0,C 180,E1 -26595.696,E2 -26595.696} C_VEL
LIN {X 0,Y 100.604,Z 327.952,A -85,B 0,C 180,E1 -26601.041,E2 -26601.041} C_VEL
LIN {X 0,Y 100.67,Z 327.937,A -85,B 0,C 180,E1 -26606.88,E2 -26606.88} C_VEL
LIN {X 0,Y 100.714,Z 327.933,A -85,B 0,C 180,E1 -26615.084,E2 -26615.084} C_VEL
LIN {X 0,Y 100.758,Z 327.933,A -85,B 0,C 180,E1 -26619.586,E2 -26619.586} C_VEL
LIN {X 0,Y 101.098,Z 327.89,A -85,B 0,C 180,E1 -26627.96,E2 -26627.96} C_VEL
LIN {X 0,Y 101.204,Z 327.875,A -85,B 0,C 180,E1 -26632.014,E2 -26632.014} C_VEL
LIN {X 0,Y 101.812,Z 327.801,A -85,B 0,C 180,E1 -26639.998,E2 -26639.998} C_VEL
LIN {X 0,Y 101.2,Z 327.878,A -85,B 0,C 180,E1 -26647.982,E2 -26647.982} C_VEL
LIN {X 0,Y 101.047,Z 327.892,A -85,B 0,C 180,E1 -26653.223,E2 -26653.223} C_VEL
LIN {X 0,Y 100.78,Z 327.923,A -85,B 0,C 180,E1 -26660.404,E2 -26660.404} C_VEL
LIN {X 0,Y 100.752,Z 327.935,A -85,B 0,C 180,E1 -26664.962,E2 -26664.962} C_VEL
LIN {X 0,Y 100.665,Z 327.946,A -85,B 0,C 180,E1 -26673.116,E2 -26673.116} C_VEL
LIN {X 0,Y 100.68,Z 328.027,A -85,B 0,C 180,E1 -26680.92,E2 -26680.92} C_VEL
LIN {X 0,Y 102.453,Z 335.698,A -85,B 0,C 180,E1 -26687.337,E2 -26687.337} C_VEL
LIN {X 0,Y 104.234,Z 343.552,A -85,B 0,C 180,E1 -26693.296,E2 -26693.296} C_VEL
LIN {X 0,Y 108.203,Z 359.664,A -85,B 0,C 180,E1 -26695.389,E2 -26695.389} C_VEL
LIN {X 0,Y 109.373,Z 387.692,A -85,B 0,C 180,E1 -26698.344,E2 -26698.344} C_VEL
LIN {X 0,Y 106.415,Z 440.118,A -85,B 0,C 180,E1 -26703.801,E2 -26703.801} C_VEL
LIN {X 0,Y 105.687,Z 449.499,A -85,B 0,C 180,E1 -26705.191,E2 -26705.191} C_VEL
LIN {X 0,Y 104.709,Z 458.949,A -85,B 0,C 180,E1 -26707.048,E2 -26707.048} C_VEL
LIN {X 0,Y 103.805,Z 467.575,A -85,B 0,C 180,E1 -26709.19,E2 -26709.19} C_VEL
LIN {X 0,Y 102.792,Z 476.943,A -85,B 0,C 180,E1 -26712.091,E2 -26712.091} C_VEL
LIN {X 0,Y 101.856,Z 485.685,A -85,B 0,C 180,E1 -26715.44,E2 -26715.44} C_VEL
LIN {X 0,Y 101.237,Z 493.392,A -85,B 0,C 180,E1 -26719.004,E2 -26719.004} C_VEL
LIN {X 0,Y 100.903,Z 500.626,A -85,B 0,C 180,E1 -26723.008,E2 -26723.008} C_VEL
LIN {X 0,Y 100.959,Z 506.751,A -85,B 0,C 180,E1 -26727.016,E2 -26727.016} C_VEL
LIN {X 0,Y 101.154,Z 512.889,A -85,B 0,C 180,E1 -26731.999,E2 -26731.999} C_VEL
LIN {X 0,Y 100.76,Z 516.736,A -85,B 0,C 180,E1 -26736.013,E2 -26736.013} C_VEL
LIN {X 0,Y 100.727,Z 522.528,A -85,B 0,C 180,E1 -26744.142,E2 -26744.142} C_VEL
LIN {X 0,Y 102.141,Z 525.82,A -85,B 0,C 180,E1 -26750.129,E2 -26750.129} C_VEL
LIN {X 0,Y 105.977,Z 528.904,A -85,B 0,C 180,E1 -26757.665,E2 -26757.665} C_VEL
LIN {X 0,Y 108.737,Z 530.056,A -85,B 0,C 180,E1 -26761.141,E2 -26761.141} C_VEL
LIN {X 0,Y 116.682,Z 531.135,A -85,B 0,C 180,E1 -26768.465,E2 -26768.465} C_VEL
LIN {X 0,Y 123.733,Z 530.886,A -85,B 0,C 180,E1 -26772.972,E2 -26772.972} C_VEL
LIN {X 0,Y 128.42,Z 530.355,A -85,B 0,C 180,E1 -26775.356,E2 -26775.356} C_VEL
LIN {X 0,Y 138.623,Z 528.118,A -85,B 0,C 180,E1 -26779.509,E2 -26779.509} C_VEL
LIN {X 0,Y 149.665,Z 524.358,A -85,B 0,C 180,E1 -26782.968,E2 -26782.968} C_VEL
LIN {X 0,Y 158.482,Z 520.507,A -85,B 0,C 180,E1 -26785.125,E2 -26785.125} C_VEL
LIN {X 0,Y 167.573,Z 515.597,A -85,B 0,C 180,E1 -26787.014,E2 -26787.014} C_VEL
LIN {X 0,Y 165.773,Z 516.516,A -85,B 0,C 180,E1 -26787.985,E2 -26787.985} C_VEL
LIN {X 0,Y 155.932,Z 520.959,A -85,B 0,C 180,E1 -26790.28,E2 -26790.28} C_VEL
LIN {X 0,Y 146.376,Z 523.958,A -85,B 0,C 180,E1 -26793,E2 -26793} C_VEL
LIN {X 0,Y 137.879,Z 525.901,A -85,B 0,C 180,E1 -26795.936,E2 -26795.936} C_VEL
LIN {X 0,Y 131.496,Z 526.626,A -85,B 0,C 180,E1 -26798.551,E2 -26798.551} C_VEL
LIN {X 0,Y 126.981,Z 526.811,A -85,B 0,C 180,E1 -26800.248,E2 -26800.248} C_VEL
LIN {X 0,Y 122.003,Z 526.779,A -85,B 0,C 180,E1 -26801.751,E2 -26801.751} C_VEL
LIN {X 0,Y 115.298,Z 526.214,A -85,B 0,C 180,E1 -26803.788,E2 -26803.788} C_VEL
LIN {X 0,Y 109.329,Z 524.952,A -85,B 0,C 180,E1 -26806.337,E2 -26806.337} C_VEL
LIN {X 0,Y 107.002,Z 524.117,A -85,B 0,C 180,E1 -26807.95,E2 -26807.95} C_VEL
LIN {X 0,Y 100.992,Z 520.628,A -85,B 0,C 180,E1 -26814.01,E2 -26814.01} C_VEL
LIN {X 0,Y 97.821,Z 517.637,A -85,B 0,C 180,E1 -26818.398,E2 -26818.398} C_VEL
LIN {X 0,Y 94.446,Z 511.906,A -85,B 0,C 180,E1 -26825.339,E2 -26825.339} C_VEL
LIN {X 0,Y 92.805,Z 506.165,A -85,B 0,C 180,E1 -26831.25,E2 -26831.25} C_VEL
LIN {X 0,Y 92.277,Z 500.031,A -85,B 0,C 180,E1 -26836.598,E2 -26836.598} C_VEL
LIN {X 0,Y 92.329,Z 493.791,A -85,B 0,C 180,E1 -26841.199,E2 -26841.199} C_VEL
LIN {X 0,Y 92.659,Z 487.397,A -85,B 0,C 180,E1 -26845.22,E2 -26845.22} C_VEL
LIN {X 0,Y 93.351,Z 478.312,A -85,B 0,C 180,E1 -26849.921,E2 -26849.921} C_VEL
LIN {X 0,Y 94.164,Z 469.88,A -85,B 0,C 180,E1 -26853.504,E2 -26853.504} C_VEL
LIN {X 0,Y 95.009,Z 461.9,A -85,B 0,C 180,E1 -26856.286,E2 -26856.286} C_VEL
LIN {X 0,Y 96.098,Z 451.846,A -85,B 0,C 180,E1 -26859.11,E2 -26859.11} C_VEL
LIN {X 0,Y 97.186,Z 440.689,A -85,B 0,C 180,E1 -26861.517,E2 -26861.517} C_VEL
LIN {X 0,Y 98.251,Z 425.866,A -85,B 0,C 180,E1 -26863.724,E2 -26863.724} C_VEL
LIN {X 0,Y 101.016,Z 381.205,A -85,B 0,C 180,E1 -26868.966,E2 -26868.966} C_VEL
LIN {X 0,Y 98.949,Z 351.704,A -85,B 0,C 180,E1 -26872.637,E2 -26872.637} C_VEL
LIN {X 0,Y 96.574,Z 341.858,A -85,B 0,C 180,E1 -26874.148,E2 -26874.148} C_VEL
LIN {X 0,Y 95.131,Z 335.123,A -85,B 0,C 180,E1 -26880.083,E2 -26880.083} C_VEL
LIN {X 0,Y 93.705,Z 328.815,A -85,B 0,C 180,E1 -26886.072,E2 -26886.072} C_VEL
LIN {X 0,Y 93.74,Z 328.809,A -85,B 0,C 180,E1 -26892.542,E2 -26892.542} C_VEL
LIN {X 0,Y 94.022,Z 328.765,A -85,B 0,C 180,E1 -26897.034,E2 -26897.034} C_VEL
LIN {X 0,Y 94.156,Z 328.756,A -85,B 0,C 180,E1 -26901.407,E2 -26901.407} C_VEL
LIN {X 0,Y 94.758,Z 328.681,A -85,B 0,C 180,E1 -26909.991,E2 -26909.991} C_VEL
LIN {X 0,Y 94.159,Z 328.756,A -85,B 0,C 180,E1 -26918.576,E2 -26918.576} C_VEL
LIN {X 0,Y 93.959,Z 328.773,A -85,B 0,C 180,E1 -26923.488,E2 -26923.488} C_VEL
LIN {X 0,Y 93.651,Z 328.81,A -85,B 0,C 180,E1 -26932.026,E2 -26932.026} C_VEL
LIN {X 0,Y 93.595,Z 328.826,A -85,B 0,C 180,E1 -26936.765,E2 -26936.765} C_VEL
LIN {X 0,Y 93.575,Z 328.829,A -85,B 0,C 180,E1 -26944.289,E2 -26944.289} C_VEL
LIN {X 0,Y 93.514,Z 328.836,A -85,B 0,C 180,E1 -26952.545,E2 -26952.545} C_VEL
LIN {X 0,Y 93.515,Z 328.828,A -85,B 0,C 180,E1 -26958.704,E2 -26958.704} C_VEL
LIN {X 0,Y 93.566,Z 328.825,A -85,B 0,C 180,E1 -26965.69,E2 -26965.69} C_VEL
LIN {X 0,Y 93.624,Z 328.819,A -85,B 0,C 180,E1 -26974.231,E2 -26974.231} C_VEL
LIN {X 0,Y 93.632,Z 328.817,A -85,B 0,C 180,E1 -26977.955,E2 -26977.955} C_VEL
LIN {X 0,Y 93.993,Z 328.774,A -85,B 0,C 180,E1 -26987.035,E2 -26987.035} C_VEL
LIN {X 0,Y 94.134,Z 328.757,A -85,B 0,C 180,E1 -26991.41,E2 -26991.41} C_VEL
LIN {X 0,Y 94.741,Z 328.682,A -85,B 0,C 180,E1 -26999.998,E2 -26999.998} C_VEL
LIN {X 0,Y 94.129,Z 328.759,A -85,B 0,C 180,E1 -27008.586,E2 -27008.586} C_VEL
LIN {X 0,Y 93.978,Z 328.774,A -85,B 0,C 180,E1 -27013.607,E2 -27013.607} C_VEL
LIN {X 0,Y 93.662,Z 328.812,A -85,B 0,C 180,E1 -27022.033,E2 -27022.033} C_VEL
LIN {X 0,Y 93.596,Z 328.824,A -85,B 0,C 180,E1 -27026.775,E2 -27026.775} C_VEL
LIN {X 0,Y 93.563,Z 328.83,A -85,B 0,C 180,E1 -27034.307,E2 -27034.307} C_VEL
LIN {X 0,Y 93.624,Z 329.017,A -85,B 0,C 180,E1 -27039.989,E2 -27039.989} C_VEL
LIN {X 0,Y 95.548,Z 337.232,A -85,B 0,C 180,E1 -27047.35,E2 -27047.35} C_VEL
LIN {X 0,Y 96.883,Z 343.26,A -85,B 0,C 180,E1 -27052.387,E2 -27052.387} C_VEL
LIN {X 0,Y 101.24,Z 360.859,A -85,B 0,C 180,E1 -27054.879,E2 -27054.879} C_VEL
LIN {X 0,Y 102.359,Z 387.023,A -85,B 0,C 180,E1 -27057.864,E2 -27057.864} C_VEL
LIN {X 0,Y 99.381,Z 438.92,A -85,B 0,C 180,E1 -27063.64,E2 -27063.64} C_VEL
LIN {X 0,Y 98.597,Z 449.192,A -85,B 0,C 180,E1 -27065.255,E2 -27065.255} C_VEL
LIN {X 0,Y 97.622,Z 458.622,A -85,B 0,C 180,E1 -27067.246,E2 -27067.246} C_VEL
LIN {X 0,Y 96.596,Z 468.404,A -85,B 0,C 180,E1 -27069.904,E2 -27069.904} C_VEL
LIN {X 0,Y 95.619,Z 477.235,A -85,B 0,C 180,E1 -27072.913,E2 -27072.913} C_VEL
LIN {X 0,Y 94.881,Z 485.014,A -85,B 0,C 180,E1 -27076.139,E2 -27076.139} C_VEL
LIN {X 0,Y 94.28,Z 493.361,A -85,B 0,C 180,E1 -27080.354,E2 -27080.354} C_VEL
LIN {X 0,Y 94.123,Z 500.46,A -85,B 0,C 180,E1 -27084.654,E2 -27084.654} C_VEL
LIN {X 0,Y 94.314,Z 506.452,A -85,B 0,C 180,E1 -27088.941,E2 -27088.941} C_VEL
LIN {X 0,Y 94.419,Z 511.407,A -85,B 0,C 180,E1 -27093.209,E2 -27093.209} C_VEL
LIN {X 0,Y 93.93,Z 516.121,A -85,B 0,C 180,E1 -27098.614,E2 -27098.614} C_VEL
LIN {X 0,Y 94.525,Z 521.81,A -85,B 0,C 180,E1 -27107.309,E2 -27107.309} C_VEL
LIN {X 0,Y 95.696,Z 524.1,A -85,B 0,C 180,E1 -27111.55,E2 -27111.55} C_VEL
LIN {X 0,Y 99.824,Z 527.626,A -85,B 0,C 180,E1 -27119.533,E2 -27119.533} C_VEL
LIN {X 0,Y 106.119,Z 529.73,A -85,B 0,C 180,E1 -27126.593,E2 -27126.593} C_VEL
LIN {X 0,Y 110.8,Z 530.442,A -85,B 0,C 180,E1 -27130.437,E2 -27130.437} C_VEL
LIN {X 0,Y 118.65,Z 530.574,A -85,B 0,C 180,E1 -27135.304,E2 -27135.304} C_VEL
LIN {X 0,Y 128.681,Z 529.469,A -85,B 0,C 180,E1 -27139.876,E2 -27139.876} C_VEL
LIN {X 0,Y 139.722,Z 526.958,A -85,B 0,C 180,E1 -27143.593,E2 -27143.593} C_VEL
LIN {X 0,Y 148.507,Z 524.144,A -85,B 0,C 180,E1 -27145.913,E2 -27145.913} C_VEL
LIN {X 0,Y 151.519,Z 522.97,A -85,B 0,C 180,E1 -27146.607,E2 -27146.607} C_VEL
LIN {X 0,Y 153.591,Z 522.071,A -85,B 0,C 180,E1 -27147.789,E2 -27147.789} C_VEL
LIN {X 0,Y 146.865,Z 524.229,A -85,B 0,C 180,E1 -27149.471,E2 -27149.471} C_VEL
LIN {X 0,Y 136.83,Z 526.378,A -85,B 0,C 180,E1 -27152.468,E2 -27152.468} C_VEL
LIN {X 0,Y 130.922,Z 527.076,A -85,B 0,C 180,E1 -27154.569,E2 -27154.569} C_VEL
LIN {X 0,Y 120.221,Z 527.154,A -85,B 0,C 180,E1 -27159.288,E2 -27159.288} C_VEL
LIN {X 0,Y 115.01,Z 526.498,A -85,B 0,C 180,E1 -27162.211,E2 -27162.211} C_VEL
LIN {X 0,Y 107.002,Z 524.117,A -85,B 0,C 180,E1 -27167.95,E2 -27167.95} C_VEL
LIN {X 0,Y 103.558,Z 522.684,A -85,B 0,C 180,E1 -27170.433,E2 -27170.433} C_VEL
LIN {X 0,Y 96.932,Z 519.466,A -85,B 0,C 180,E1 -27174.254,E2 -27174.254} C_VEL
LIN {X 0,Y 91.012,Z 515.482,A -85,B 0,C 180,E1 -27178.471,E2 -27178.471} C_VEL
LIN {X 0,Y 88.811,Z 512.732,A -85,B 0,C 180,E1 -27181.509,E2 -27181.509} C_VEL
LIN {X 0,Y 86.525,Z 506.657,A -85,B 0,C 180,E1 -27188.175,E2 -27188.175} C_VEL
LIN {X 0,Y 85.572,Z 500.215,A -85,B 0,C 180,E1 -27194.267,E2 -27194.267} C_VEL
LIN {X 0,Y 85.437,Z 494.12,A -85,B 0,C 180,E1 -27199.213,E2 -27199.213} C_VEL
LIN {X 0,Y 85.721,Z 486.691,A -85,B 0,C 180,E1 -27204.203,E2 -27204.203} C_VEL
LIN {X 0,Y 86.275,Z 478.67,A -85,B 0,C 180,E1 -27208.676,E2 -27208.676} C_VEL
LIN {X 0,Y 87.003,Z 470.751,A -85,B 0,C 180,E1 -27212.358,E2 -27212.358} C_VEL
LIN {X 0,Y 88.006,Z 460.809,A -85,B 0,C 180,E1 -27216.118,E2 -27216.118} C_VEL
LIN {X 0,Y 89.176,Z 449.546,A -85,B 0,C 180,E1 -27219.454,E2 -27219.454} C_VEL
LIN {X 0,Y 90.479,Z 435.91,A -85,B 0,C 180,E1 -27222.348,E2 -27222.348} C_VEL
LIN {X 0,Y 92.163,Z 409.622,A -85,B 0,C 180,E1 -27225.941,E2 -27225.941} C_VEL
LIN {X 0,Y 93.939,Z 381.421,A -85,B 0,C 180,E1 -27229.459,E2 -27229.459} C_VEL
LIN {X 0,Y 91.938,Z 352.596,A -85,B 0,C 180,E1 -27233.323,E2 -27233.323} C_VEL
LIN {X 0,Y 89.386,Z 341.923,A -85,B 0,C 180,E1 -27235.069,E2 -27235.069} C_VEL
LIN {X 0,Y 87.642,Z 334.029,A -85,B 0,C 180,E1 -27242.655,E2 -27242.655} C_VEL
LIN {X 0,Y 86.645,Z 329.693,A -85,B 0,C 180,E1 -27247.331,E2 -27247.331} C_VEL
LIN {X 0,Y 86.872,Z 329.654,A -85,B 0,C 180,E1 -27256.134,E2 -27256.134} C_VEL
LIN {X 0,Y 87.062,Z 329.64,A -85,B 0,C 180,E1 -27260.7,E2 -27260.7} C_VEL
LIN {X 0,Y 87.687,Z 329.562,A -85,B 0,C 180,E1 -27269.991,E2 -27269.991} C_VEL
LIN {X 0,Y 87.062,Z 329.639,A -85,B 0,C 180,E1 -27279.281,E2 -27279.281} C_VEL
LIN {X 0,Y 86.859,Z 329.659,A -85,B 0,C 180,E1 -27284.037,E2 -27284.037} C_VEL
LIN {X 0,Y 86.597,Z 329.696,A -85,B 0,C 180,E1 -27288.931,E2 -27288.931} C_VEL
LIN {X 0,Y 86.561,Z 329.703,A -85,B 0,C 180,E1 -27296.728,E2 -27296.728} C_VEL
LIN {X 0,Y 86.492,Z 329.712,A -85,B 0,C 180,E1 -27305.649,E2 -27305.649} C_VEL
LIN {X 0,Y 86.438,Z 329.717,A -85,B 0,C 180,E1 -27312.962,E2 -27312.962} C_VEL
LIN {X 0,Y 86.437,Z 329.711,A -85,B 0,C 180,E1 -27319.42,E2 -27319.42} C_VEL
LIN {X 0,Y 86.509,Z 329.705,A -85,B 0,C 180,E1 -27325.339,E2 -27325.339} C_VEL
LIN {X 0,Y 86.547,Z 329.703,A -85,B 0,C 180,E1 -27333.252,E2 -27333.252} C_VEL
LIN {X 0,Y 86.576,Z 329.7,A -85,B 0,C 180,E1 -27341.049,E2 -27341.049} C_VEL
LIN {X 0,Y 86.838,Z 329.66,A -85,B 0,C 180,E1 -27346.151,E2 -27346.151} C_VEL
LIN {X 0,Y 87.038,Z 329.642,A -85,B 0,C 180,E1 -27350.704,E2 -27350.704} C_VEL
LIN {X 0,Y 87.671,Z 329.563,A -85,B 0,C 180,E1 -27359.998,E2 -27359.998} C_VEL
LIN {X 0,Y 87.023,Z 329.642,A -85,B 0,C 180,E1 -27369.293,E2 -27369.293} C_VEL
LIN {X 0,Y 86.87,Z 329.661,A -85,B 0,C 180,E1 -27374.044,E2 -27374.044} C_VEL
LIN {X 0,Y 86.601,Z 329.693,A -85,B 0,C 180,E1 -27378.94,E2 -27378.94} C_VEL
LIN {X 0,Y 86.56,Z 329.7,A -85,B 0,C 180,E1 -27386.765,E2 -27386.765} C_VEL
LIN {X 0,Y 86.485,Z 329.71,A -85,B 0,C 180,E1 -27395.671,E2 -27395.671} C_VEL
LIN {X 0,Y 86.541,Z 329.869,A -85,B 0,C 180,E1 -27398.819,E2 -27398.819} C_VEL
LIN {X 0,Y 88.214,Z 337.003,A -85,B 0,C 180,E1 -27405.806,E2 -27405.806} C_VEL
LIN {X 0,Y 89.625,Z 343.209,A -85,B 0,C 180,E1 -27411.467,E2 -27411.467} C_VEL
LIN {X 0,Y 94.289,Z 362.5,A -85,B 0,C 180,E1 -27414.378,E2 -27414.378} C_VEL
LIN {X 0,Y 95.275,Z 387.441,A -85,B 0,C 180,E1 -27417.436,E2 -27417.436} C_VEL
LIN {X 0,Y 92.303,Z 438.545,A -85,B 0,C 180,E1 -27423.593,E2 -27423.593} C_VEL
LIN {X 0,Y 91.516,Z 448.709,A -85,B 0,C 180,E1 -27425.331,E2 -27425.331} C_VEL
LIN {X 0,Y 90.46,Z 459.11,A -85,B 0,C 180,E1 -27427.757,E2 -27427.757} C_VEL
LIN {X 0,Y 89.37,Z 469.57,A -85,B 0,C 180,E1 -27430.949,E2 -27430.949} C_VEL
LIN {X 0,Y 88.29,Z 480.111,A -85,B 0,C 180,E1 -27435.081,E2 -27435.081} C_VEL
LIN {X 0,Y 87.482,Z 491.274,A -85,B 0,C 180,E1 -27440.764,E2 -27440.764} C_VEL
LIN {X 0,Y 87.365,Z 498.621,A -85,B 0,C 180,E1 -27445.396,E2 -27445.396} C_VEL
LIN {X 0,Y 87.714,Z 506.119,A -85,B 0,C 180,E1 -27451.157,E2 -27451.157} C_VEL
LIN {X 0,Y 87.772,Z 509.812,A -85,B 0,C 180,E1 -27454.602,E2 -27454.602} C_VEL
LIN {X 0,Y 87.251,Z 515.314,A -85,B 0,C 180,E1 -27461.626,E2 -27461.626} C_VEL
LIN {X 0,Y 88.626,Z 521.066,A -85,B 0,C 180,E1 -27470.914,E2 -27470.914} C_VEL
LIN {X 0,Y 91.264,Z 524.349,A -85,B 0,C 180,E1 -27477.526,E2 -27477.526} C_VEL
LIN {X 0,Y 96.997,Z 527.502,A -85,B 0,C 180,E1 -27485.432,E2 -27485.432} C_VEL
LIN {X 0,Y 104.576,Z 529.344,A -85,B 0,C 180,E1 -27492.231,E2 -27492.231} C_VEL
LIN {X 0,Y 109.004,Z 529.899,A -85,B 0,C 180,E1 -27495.177,E2 -27495.177} C_VEL
LIN {X 0,Y 118.898,Z 529.878,A -85,B 0,C 180,E1 -27500.217,E2 -27500.217} C_VEL
LIN {X 0,Y 129.872,Z 528.529,A -85,B 0,C 180,E1 -27504.267,E2 -27504.267} C_VEL
LIN {X 0,Y 138.029,Z 526.828,A -85,B 0,C 180,E1 -27506.633,E2 -27506.633} C_VEL
LIN {X 0,Y 140.186,Z 526.121,A -85,B 0,C 180,E1 -27507.901,E2 -27507.901} C_VEL
LIN {X 0,Y 136.349,Z 526.873,A -85,B 0,C 180,E1 -27508.975,E2 -27508.975} C_VEL
LIN {X 0,Y 127.713,Z 527.796,A -85,B 0,C 180,E1 -27511.702,E2 -27511.702} C_VEL
LIN {X 0,Y 117.983,Z 527.701,A -85,B 0,C 180,E1 -27515.553,E2 -27515.553} C_VEL
LIN {X 0,Y 112.838,Z 527.104,A -85,B 0,C 180,E1 -27518.058,E2 -27518.058} C_VEL
LIN {X 0,Y 103.111,Z 524.566,A -85,B 0,C 180,E1 -27524.181,E2 -27524.181} C_VEL
LIN {X 0,Y 97.041,Z 521.475,A -85,B 0,C 180,E1 -27529.571,E2 -27529.571} C_VEL
LIN {X 0,Y 92.104,Z 517.34,A -85,B 0,C 180,E1 -27535.626,E2 -27535.626} C_VEL
LIN {X 0,Y 88.811,Z 512.732,A -85,B 0,C 180,E1 -27541.509,E2 -27541.509} C_VEL
LIN {X 0,Y 86.972,Z 509.86,A -85,B 0,C 180,E1 -27544.586,E2 -27544.586} C_VEL
LIN {X 0,Y 84.578,Z 506.58,A -85,B 0,C 180,E1 -27547.458,E2 -27547.458} C_VEL
LIN {X 0,Y 79.455,Z 497.782,A -85,B 0,C 180,E1 -27554.171,E2 -27554.171} C_VEL
LIN {X 0,Y 78.678,Z 493.671,A -85,B 0,C 180,E1 -27557.318,E2 -27557.318} C_VEL
LIN {X 0,Y 78.864,Z 485.984,A -85,B 0,C 180,E1 -27562.95,E2 -27562.95} C_VEL
LIN {X 0,Y 79.296,Z 478.346,A -85,B 0,C 180,E1 -27567.577,E2 -27567.577} C_VEL
LIN {X 0,Y 80.01,Z 469.831,A -85,B 0,C 180,E1 -27571.808,E2 -27571.808} C_VEL
LIN {X 0,Y 80.839,Z 461.642,A -85,B 0,C 180,E1 -27575.17,E2 -27575.17} C_VEL
LIN {X 0,Y 81.979,Z 450.559,A -85,B 0,C 180,E1 -27578.794,E2 -27578.794} C_VEL
LIN {X 0,Y 83.282,Z 436.858,A -85,B 0,C 180,E1 -27582.041,E2 -27582.041} C_VEL
LIN {X 0,Y 84.87,Z 412.072,A -85,B 0,C 180,E1 -27585.796,E2 -27585.796} C_VEL
LIN {X 0,Y 86.92,Z 382.22,A -85,B 0,C 180,E1 -27589.878,E2 -27589.878} C_VEL
LIN {X 0,Y 85.081,Z 354.095,A -85,B 0,C 180,E1 -27593.938,E2 -27593.938} C_VEL
LIN {X 0,Y 82.117,Z 341.92,A -85,B 0,C 180,E1 -27596.191,E2 -27596.191} C_VEL
LIN {X 0,Y 80.441,Z 334.376,A -85,B 0,C 180,E1 -27604.089,E2 -27604.089} C_VEL
LIN {X 0,Y 79.579,Z 330.573,A -85,B 0,C 180,E1 -27608.627,E2 -27608.627} C_VEL
LIN {X 0,Y 79.795,Z 330.536,A -85,B 0,C 180,E1 -27615.669,E2 -27615.669} C_VEL
LIN {X 0,Y 79.939,Z 330.527,A -85,B 0,C 180,E1 -27619.863,E2 -27619.863} C_VEL
LIN {X 0,Y 80.617,Z 330.443,A -85,B 0,C 180,E1 -27629.99,E2 -27629.99} C_VEL
LIN {X 0,Y 79.937,Z 330.525,A -85,B 0,C 180,E1 -27640.116,E2 -27640.116} C_VEL
LIN {X 0,Y 79.687,Z 330.557,A -85,B 0,C 180,E1 -27645.33,E2 -27645.33} C_VEL
LIN {X 0,Y 79.475,Z 330.577,A -85,B 0,C 180,E1 -27650.702,E2 -27650.702} C_VEL
LIN {X 0,Y 79.462,Z 330.585,A -85,B 0,C 180,E1 -27657.81,E2 -27657.81} C_VEL
LIN {X 0,Y 79.363,Z 330.593,A -85,B 0,C 180,E1 -27662.08,E2 -27662.08} C_VEL
LIN {X 0,Y 79.352,Z 330.593,A -85,B 0,C 180,E1 -27668.297,E2 -27668.297} C_VEL
LIN {X 0,Y 79.34,Z 330.601,A -85,B 0,C 180,E1 -27675.105,E2 -27675.105} C_VEL
LIN {X 0,Y 79.367,Z 330.599,A -85,B 0,C 180,E1 -27682.816,E2 -27682.816} C_VEL
LIN {X 0,Y 79.353,Z 330.592,A -85,B 0,C 180,E1 -27687.897,E2 -27687.897} C_VEL
LIN {X 0,Y 79.488,Z 330.58,A -85,B 0,C 180,E1 -27693.76,E2 -27693.76} C_VEL
LIN {X 0,Y 79.456,Z 330.586,A -85,B 0,C 180,E1 -27699.277,E2 -27699.277} C_VEL
LIN {X 0,Y 79.764,Z 330.54,A -85,B 0,C 180,E1 -27705.681,E2 -27705.681} C_VEL
LIN {X 0,Y 79.912,Z 330.531,A -85,B 0,C 180,E1 -27709.867,E2 -27709.867} C_VEL
LIN {X 0,Y 80.601,Z 330.444,A -85,B 0,C 180,E1 -27719.997,E2 -27719.997} C_VEL
LIN {X 0,Y 79.911,Z 330.526,A -85,B 0,C 180,E1 -27730.128,E2 -27730.128} C_VEL
LIN {X 0,Y 79.703,Z 330.556,A -85,B 0,C 180,E1 -27735.336,E2 -27735.336} C_VEL
LIN {X 0,Y 79.477,Z 330.576,A -85,B 0,C 180,E1 -27740.712,E2 -27740.712} C_VEL
LIN {X 0,Y 79.457,Z 330.582,A -85,B 0,C 180,E1 -27747.843,E2 -27747.843} C_VEL
LIN {X 0,Y 79.442,Z 330.737,A -85,B 0,C 180,E1 -27757.525,E2 -27757.525} C_VEL
LIN {X 0,Y 80.863,Z 336.82,A -85,B 0,C 180,E1 -27764.047,E2 -27764.047} C_VEL
LIN {X 0,Y 82.356,Z 343.216,A -85,B 0,C 180,E1 -27770.432,E2 -27770.432} C_VEL
LIN {X 0,Y 87.304,Z 363.219,A -85,B 0,C 180,E1 -27773.748,E2 -27773.748} C_VEL
LIN {X 0,Y 88.234,Z 387.513,A -85,B 0,C 180,E1 -27776.982,E2 -27776.982} C_VEL
LIN {X 0,Y 85.224,Z 438.329,A -85,B 0,C 180,E1 -27783.702,E2 -27783.702} C_VEL
LIN {X 0,Y 84.502,Z 447.797,A -85,B 0,C 180,E1 -27785.441,E2 -27785.441} C_VEL
LIN {X 0,Y 83.468,Z 458,A -85,B 0,C 180,E1 -27787.982,E2 -27787.982} C_VEL
LIN {X 0,Y 82.533,Z 467.298,A -85,B 0,C 180,E1 -27790.972,E2 -27790.972} C_VEL
LIN {X 0,Y 81.669,Z 475.402,A -85,B 0,C 180,E1 -27794.204,E2 -27794.204} C_VEL
LIN {X 0,Y 80.938,Z 484.659,A -85,B 0,C 180,E1 -27798.745,E2 -27798.745} C_VEL
LIN {X 0,Y 80.63,Z 491.088,A -85,B 0,C 180,E1 -27802.498,E2 -27802.498} C_VEL
LIN {X 0,Y 80.708,Z 498.321,A -85,B 0,C 180,E1 -27807.515,E2 -27807.515} C_VEL
LIN {X 0,Y 81.12,Z 504.368,A -85,B 0,C 180,E1 -27812.493,E2 -27812.493} C_VEL
LIN {X 0,Y 81.177,Z 507.935,A -85,B 0,C 180,E1 -27816.222,E2 -27816.222} C_VEL
LIN {X 0,Y 80.811,Z 512.733,A -85,B 0,C 180,E1 -27822.567,E2 -27822.567} C_VEL
LIN {X 0,Y 81.714,Z 517.499,A -85,B 0,C 180,E1 -27830.131,E2 -27830.131} C_VEL
LIN {X 0,Y 84.105,Z 521.313,A -85,B 0,C 180,E1 -27837.369,E2 -27837.369} C_VEL
LIN {X 0,Y 88.032,Z 524.405,A -85,B 0,C 180,E1 -27843.983,E2 -27843.983} C_VEL
LIN {X 0,Y 91.418,Z 526.057,A -85,B 0,C 180,E1 -27847.96,E2 -27847.96} C_VEL
LIN {X 0,Y 100.517,Z 528.505,A -85,B 0,C 180,E1 -27855.641,E2 -27855.641} C_VEL
LIN {X 0,Y 109.175,Z 529.363,A -85,B 0,C 180,E1 -27860.582,E2 -27860.582} C_VEL
LIN {X 0,Y 120.037,Z 529.124,A -85,B 0,C 180,E1 -27865.056,E2 -27865.056} C_VEL
LIN {X 0,Y 125.866,Z 528.592,A -85,B 0,C 180,E1 -27866.886,E2 -27866.886} C_VEL
LIN {X 0,Y 127.11,Z 528.341,A -85,B 0,C 180,E1 -27867.986,E2 -27867.986} C_VEL
LIN {X 0,Y 117.225,Z 528.331,A -85,B 0,C 180,E1 -27871.341,E2 -27871.341} C_VEL
LIN {X 0,Y 108.44,Z 527.285,A -85,B 0,C 180,E1 -27875.145,E2 -27875.145} C_VEL
LIN {X 0,Y 100.629,Z 525.273,A -85,B 0,C 180,E1 -27879.564,E2 -27879.564} C_VEL
LIN {X 0,Y 93.679,Z 522.261,A -85,B 0,C 180,E1 -27884.82,E2 -27884.82} C_VEL
LIN {X 0,Y 87.912,Z 518.253,A -85,B 0,C 180,E1 -27890.802,E2 -27890.802} C_VEL
LIN {X 0,Y 83.551,Z 513.302,A -85,B 0,C 180,E1 -27897.351,E2 -27897.351} C_VEL
LIN {X 0,Y 80.813,Z 507.958,A -85,B 0,C 180,E1 -27903.742,E2 -27903.742} C_VEL
LIN {X 0,Y 79.182,Z 501.687,A -85,B 0,C 180,E1 -27910.228,E2 -27910.228} C_VEL
LIN {X 0,Y 78.685,Z 494.222,A -85,B 0,C 180,E1 -27916.878,E2 -27916.878} C_VEL
LIN {X 0,Y 78.678,Z 493.671,A -85,B 0,C 180,E1 -27917.318,E2 -27917.318} C_VEL
LIN {X 0,Y 78.089,Z 489.637,A -85,B 0,C 180,E1 -27920.282,E2 -27920.282} C_VEL
LIN {X 0,Y 76.749,Z 485.147,A -85,B 0,C 180,E1 -27922.958,E2 -27922.958} C_VEL
LIN {X 0,Y 73.373,Z 473.786,A -85,B 0,C 180,E1 -27928.76,E2 -27928.76} C_VEL
LIN {X 0,Y 73.076,Z 468.55,A -85,B 0,C 180,E1 -27931.25,E2 -27931.25} C_VEL
LIN {X 0,Y 74.182,Z 456.711,A -85,B 0,C 180,E1 -27936.312,E2 -27936.312} C_VEL
LIN {X 0,Y 75.322,Z 445.029,A -85,B 0,C 180,E1 -27939.906,E2 -27939.906} C_VEL
LIN {X 0,Y 76.292,Z 435.302,A -85,B 0,C 180,E1 -27942.152,E2 -27942.152} C_VEL
LIN {X 0,Y 78.72,Z 398.299,A -85,B 0,C 180,E1 -27948.036,E2 -27948.036} C_VEL
LIN {X 0,Y 79.804,Z 381.761,A -85,B 0,C 180,E1 -27950.471,E2 -27950.471} C_VEL
LIN {X 0,Y 78.077,Z 355.022,A -85,B 0,C 180,E1 -27954.696,E2 -27954.696} C_VEL
LIN {X 0,Y 74.872,Z 342.01,A -85,B 0,C 180,E1 -27957.277,E2 -27957.277} C_VEL
LIN {X 0,Y 73.207,Z 334.55,A -85,B 0,C 180,E1 -27965.911,E2 -27965.911} C_VEL
LIN {X 0,Y 72.514,Z 331.453,A -85,B 0,C 180,E1 -27969.792,E2 -27969.792} C_VEL
LIN {X 0,Y 72.831,Z 331.41,A -85,B 0,C 180,E1 -27978.862,E2 -27978.862} C_VEL
LIN {X 0,Y 73.545,Z 331.324,A -85,B 0,C 180,E1 -27989.989,E2 -27989.989} C_VEL
LIN {X 0,Y 72.828,Z 331.408,A -85,B 0,C 180,E1 -28001.116,E2 -28001.116} C_VEL
LIN {X 0,Y 72.504,Z 331.454,A -85,B 0,C 180,E1 -28006.892,E2 -28006.892} C_VEL
LIN {X 0,Y 72.364,Z 331.463,A -85,B 0,C 180,E1 -28012.845,E2 -28012.845} C_VEL
LIN {X 0,Y 72.352,Z 331.466,A -85,B 0,C 180,E1 -28019.041,E2 -28019.041} C_VEL
LIN {X 0,Y 72.281,Z 331.481,A -85,B 0,C 180,E1 -28025.671,E2 -28025.671} C_VEL
LIN {X 0,Y 72.214,Z 331.489,A -85,B 0,C 180,E1 -28032.921,E2 -28032.921} C_VEL
LIN {X 0,Y 72.274,Z 331.48,A -85,B 0,C 180,E1 -28041.046,E2 -28041.046} C_VEL
LIN {X 0,Y 72.274,Z 331.481,A -85,B 0,C 180,E1 -28044.303,E2 -28044.303} C_VEL
LIN {X 0,Y 72.342,Z 331.473,A -85,B 0,C 180,E1 -28050.935,E2 -28050.935} C_VEL
LIN {X 0,Y 72.347,Z 331.465,A -85,B 0,C 180,E1 -28057.131,E2 -28057.131} C_VEL
LIN {X 0,Y 72.657,Z 331.424,A -85,B 0,C 180,E1 -28065.239,E2 -28065.239} C_VEL
LIN {X 0,Y 72.804,Z 331.416,A -85,B 0,C 180,E1 -28068.865,E2 -28068.865} C_VEL
LIN {X 0,Y 73.528,Z 331.325,A -85,B 0,C 180,E1 -28079.997,E2 -28079.997} C_VEL
LIN {X 0,Y 72.809,Z 331.407,A -85,B 0,C 180,E1 -28091.128,E2 -28091.128} C_VEL
LIN {X 0,Y 72.54,Z 331.449,A -85,B 0,C 180,E1 -28096.894,E2 -28096.894} C_VEL
LIN {X 0,Y 72.364,Z 331.467,A -85,B 0,C 180,E1 -28102.857,E2 -28102.857} C_VEL
LIN {X 0,Y 72.338,Z 331.464,A -85,B 0,C 180,E1 -28109.06,E2 -28109.06} C_VEL
LIN {X 0,Y 72.348,Z 331.602,A -85,B 0,C 180,E1 -28116.063,E2 -28116.063} C_VEL
LIN {X 0,Y 73.868,Z 337.981,A -85,B 0,C 180,E1 -28123.609,E2 -28123.609} C_VEL
LIN {X 0,Y 75.062,Z 343.054,A -85,B 0,C 180,E1 -28129.199,E2 -28129.199} C_VEL
LIN {X 0,Y 80.346,Z 364.709,A -85,B 0,C 180,E1 -28133.214,E2 -28133.214} C_VEL
LIN {X 0,Y 81.117,Z 388.225,A -85,B 0,C 180,E1 -28136.614,E2 -28136.614} C_VEL
LIN {X 0,Y 78.139,Z 438.204,A -85,B 0,C 180,E1 -28143.849,E2 -28143.849} C_VEL
LIN {X 0,Y 77.342,Z 448.334,A -85,B 0,C 180,E1 -28145.927,E2 -28145.927} C_VEL
LIN {X 0,Y 76.293,Z 458.484,A -85,B 0,C 180,E1 -28148.762,E2 -28148.762} C_VEL
LIN {X 0,Y 75.479,Z 467.065,A -85,B 0,C 180,E1 -28151.835,E2 -28151.835} C_VEL
LIN {X 0,Y 74.55,Z 477.043,A -85,B 0,C 180,E1 -28156.381,E2 -28156.381} C_VEL
LIN {X 0,Y 73.99,Z 485.428,A -85,B 0,C 180,E1 -28161.133,E2 -28161.133} C_VEL
LIN {X 0,Y 73.932,Z 492.531,A -85,B 0,C 180,E1 -28165.923,E2 -28165.923} C_VEL
LIN {X 0,Y 74.386,Z 499.41,A -85,B 0,C 180,E1 -28171.364,E2 -28171.364} C_VEL
LIN {X 0,Y 74.713,Z 503.786,A -85,B 0,C 180,E1 -28175.408,E2 -28175.408} C_VEL
LIN {X 0,Y 74.465,Z 508.179,A -85,B 0,C 180,E1 -28180.89,E2 -28180.89} C_VEL
LIN {X 0,Y 75.456,Z 515.15,A -85,B 0,C 180,E1 -28191.883,E2 -28191.883} C_VEL
LIN {X 0,Y 79.398,Z 520.432,A -85,B 0,C 180,E1 -28202.088,E2 -28202.088} C_VEL
LIN {X 0,Y 82.419,Z 522.595,A -85,B 0,C 180,E1 -28206.656,E2 -28206.656} C_VEL
LIN {X 0,Y 90.123,Z 525.93,A -85,B 0,C 180,E1 -28214.582,E2 -28214.582} C_VEL
LIN {X 0,Y 99.588,Z 527.947,A -85,B 0,C 180,E1 -28220.927,E2 -28220.927} C_VEL
LIN {X 0,Y 110.382,Z 528.775,A -85,B 0,C 180,E1 -28225.868,E2 -28225.868} C_VEL
LIN {X 0,Y 112.409,Z 528.783,A -85,B 0,C 180,E1 -28226.624,E2 -28226.624} C_VEL
LIN {X 0,Y 114.278,Z 528.68,A -85,B 0,C 180,E1 -28228.059,E2 -28228.059} C_VEL
LIN {X 0,Y 102.798,Z 526.919,A -85,B 0,C 180,E1 -28232.726,E2 -28232.726} C_VEL
LIN {X 0,Y 98.887,Z 525.968,A -85,B 0,C 180,E1 -28234.761,E2 -28234.761} C_VEL
LIN {X 0,Y 91.261,Z 523.092,A -85,B 0,C 180,E1 -28239.616,E2 -28239.616} C_VEL
LIN {X 0,Y 84.439,Z 519.096,A -85,B 0,C 180,E1 -28245.543,E2 -28245.543} C_VEL
LIN {X 0,Y 79.09,Z 514.192,A -85,B 0,C 180,E1 -28252.239,E2 -28252.239} C_VEL
LIN {X 0,Y 75.084,Z 507.894,A -85,B 0,C 180,E1 -28260.003,E2 -28260.003} C_VEL
LIN {X 0,Y 72.961,Z 501.686,A -85,B 0,C 180,E1 -28266.919,E2 -28266.919} C_VEL
LIN {X 0,Y 72.141,Z 495.547,A -85,B 0,C 180,E1 -28273.017,E2 -28273.017} C_VEL
LIN {X 0,Y 71.979,Z 487.102,A -85,B 0,C 180,E1 -28279.986,E2 -28279.986} C_VEL
LIN {X 0,Y 72.245,Z 479.484,A -85,B 0,C 180,E1 -28285.192,E2 -28285.192} C_VEL
LIN {X 0,Y 72.816,Z 471.649,A -85,B 0,C 180,E1 -28289.685,E2 -28289.685} C_VEL
LIN {X 0,Y 73.076,Z 468.55,A -85,B 0,C 180,E1 -28291.25,E2 -28291.25} C_VEL
LIN {X 0,Y 72.806,Z 463.423,A -85,B 0,C 180,E1 -28293.517,E2 -28293.517} C_VEL
LIN {X 0,Y 70.775,Z 454.515,A -85,B 0,C 180,E1 -28296.612,E2 -28296.612} C_VEL
LIN {X 0,Y 68.839,Z 445.422,A -85,B 0,C 180,E1 -28299.339,E2 -28299.339} C_VEL
LIN {X 0,Y 68.789,Z 439.601,A -85,B 0,C 180,E1 -28300.897,E2 -28300.897} C_VEL
LIN {X 0,Y 70.109,Z 421.73,A -85,B 0,C 180,E1 -28304.443,E2 -28304.443} C_VEL
LIN {X 0,Y 72.73,Z 381.914,A -85,B 0,C 180,E1 -28311.076,E2 -28311.076} C_VEL
LIN {X 0,Y 71.072,Z 355.918,A -85,B 0,C 180,E1 -28315.554,E2 -28315.554} C_VEL
LIN {X 0,Y 67.63,Z 342.036,A -85,B 0,C 180,E1 -28318.685,E2 -28318.685} C_VEL
LIN {X 0,Y 66.232,Z 335.895,A -85,B 0,C 180,E1 -28326.541,E2 -28326.541} C_VEL
LIN {X 0,Y 65.454,Z 332.332,A -85,B 0,C 180,E1 -28331.735,E2 -28331.735} C_VEL
LIN {X 0,Y 65.726,Z 332.29,A -85,B 0,C 180,E1 -28337.64,E2 -28337.64} C_VEL
LIN {X 0,Y 66.444,Z 332.208,A -85,B 0,C 180,E1 -28349.988,E2 -28349.988} C_VEL
LIN {X 0,Y 65.721,Z 332.289,A -85,B 0,C 180,E1 -28362.336,E2 -28362.336} C_VEL
LIN {X 0,Y 65.335,Z 332.344,A -85,B 0,C 180,E1 -28368.812,E2 -28368.812} C_VEL
LIN {X 0,Y 65.213,Z 332.362,A -85,B 0,C 180,E1 -28375.52,E2 -28375.52} C_VEL
LIN {X 0,Y 65.161,Z 332.363,A -85,B 0,C 180,E1 -28382.616,E2 -28382.616} C_VEL
LIN {X 0,Y 65.157,Z 332.361,A -85,B 0,C 180,E1 -28390.966,E2 -28390.966} C_VEL
LIN {X 0,Y 65.175,Z 332.359,A -85,B 0,C 180,E1 -28399.68,E2 -28399.68} C_VEL
LIN {X 0,Y 65.208,Z 332.358,A -85,B 0,C 180,E1 -28409.533,E2 -28409.533} C_VEL
LIN {X 0,Y 65.198,Z 332.357,A -85,B 0,C 180,E1 -28414.454,E2 -28414.454} C_VEL
LIN {X 0,Y 65.56,Z 332.308,A -85,B 0,C 180,E1 -28424.684,E2 -28424.684} C_VEL
LIN {X 0,Y 65.698,Z 332.299,A -85,B 0,C 180,E1 -28427.643,E2 -28427.643} C_VEL
LIN {X 0,Y 66.427,Z 332.209,A -85,B 0,C 180,E1 -28439.997,E2 -28439.997} C_VEL
LIN {X 0,Y 65.712,Z 332.29,A -85,B 0,C 180,E1 -28452.348,E2 -28452.348} C_VEL
LIN {X 0,Y 65.349,Z 332.339,A -85,B 0,C 180,E1 -28458.819,E2 -28458.819} C_VEL
LIN {X 0,Y 65.206,Z 332.363,A -85,B 0,C 180,E1 -28465.535,E2 -28465.535} C_VEL
LIN {X 0,Y 65.176,Z 332.366,A -85,B 0,C 180,E1 -28473.544,E2 -28473.544} C_VEL
LIN {X 0,Y 65.228,Z 332.575,A -85,B 0,C 180,E1 -28474.444,E2 -28474.444} C_VEL
LIN {X 0,Y 66.58,Z 337.911,A -85,B 0,C 180,E1 -28481.569,E2 -28481.569} C_VEL
LIN {X 0,Y 67.769,Z 343.081,A -85,B 0,C 180,E1 -28487.924,E2 -28487.924} C_VEL
LIN {X 0,Y 73.218,Z 364.803,A -85,B 0,C 180,E1 -28492.361,E2 -28492.361} C_VEL
LIN {X 0,Y 74.105,Z 387.559,A -85,B 0,C 180,E1 -28495.976,E2 -28495.976} C_VEL
LIN {X 0,Y 71.031,Z 438.195,A -85,B 0,C 180,E1 -28504.151,E2 -28504.151} C_VEL
LIN {X 0,Y 70.247,Z 448.06,A -85,B 0,C 180,E1 -28506.425,E2 -28506.425} C_VEL
LIN {X 0,Y 69.35,Z 457.192,A -85,B 0,C 180,E1 -28509.24,E2 -28509.24} C_VEL
LIN {X 0,Y 68.503,Z 466.387,A -85,B 0,C 180,E1 -28512.859,E2 -28512.859} C_VEL
LIN {X 0,Y 67.751,Z 475.323,A -85,B 0,C 180,E1 -28517.279,E2 -28517.279} C_VEL
LIN {X 0,Y 67.339,Z 482.812,A -85,B 0,C 180,E1 -28521.762,E2 -28521.762} C_VEL
LIN {X 0,Y 67.304,Z 490.219,A -85,B 0,C 180,E1 -28527.02,E2 -28527.02} C_VEL
LIN {X 0,Y 67.896,Z 497.381,A -85,B 0,C 180,E1 -28532.978,E2 -28532.978} C_VEL
LIN {X 0,Y 68.323,Z 501.743,A -85,B 0,C 180,E1 -28537.399,E2 -28537.399} C_VEL
LIN {X 0,Y 68.146,Z 506.106,A -85,B 0,C 180,E1 -28543.428,E2 -28543.428} C_VEL
LIN {X 0,Y 68.804,Z 510.88,A -85,B 0,C 180,E1 -28551.075,E2 -28551.075} C_VEL
LIN {X 0,Y 71.165,Z 515.545,A -85,B 0,C 180,E1 -28559.599,E2 -28559.599} C_VEL
LIN {X 0,Y 75.336,Z 519.444,A -85,B 0,C 180,E1 -28567.337,E2 -28567.337} C_VEL
LIN {X 0,Y 80.972,Z 522.649,A -85,B 0,C 180,E1 -28573.985,E2 -28573.985} C_VEL
LIN {X 0,Y 91.907,Z 526.021,A -85,B 0,C 180,E1 -28582.287,E2 -28582.287} C_VEL
LIN {X 0,Y 100.83,Z 527.507,A -85,B 0,C 180,E1 -28586.77,E2 -28586.77} C_VEL
LIN {X 0,Y 101.777,Z 527.465,A -85,B 0,C 180,E1 -28588.128,E2 -28588.128} C_VEL
LIN {X 0,Y 97.333,Z 526.445,A -85,B 0,C 180,E1 -28590.058,E2 -28590.058} C_VEL
LIN {X 0,Y 89.336,Z 523.728,A -85,B 0,C 180,E1 -28594.365,E2 -28594.365} C_VEL
LIN {X 0,Y 81.767,Z 519.887,A -85,B 0,C 180,E1 -28599.894,E2 -28599.894} C_VEL
LIN {X 0,Y 75.362,Z 514.975,A -85,B 0,C 180,E1 -28606.521,E2 -28606.521} C_VEL
LIN {X 0,Y 70.355,Z 508.965,A -85,B 0,C 180,E1 -28614.27,E2 -28614.27} C_VEL
LIN {X 0,Y 67.47,Z 502.925,A -85,B 0,C 180,E1 -28621.495,E2 -28621.495} C_VEL
LIN {X 0,Y 65.788,Z 495.777,A -85,B 0,C 180,E1 -28629.224,E2 -28629.224} C_VEL
LIN {X 0,Y 65.295,Z 487.865,A -85,B 0,C 180,E1 -28636.659,E2 -28636.659} C_VEL
LIN {X 0,Y 65.353,Z 480.867,A -85,B 0,C 180,E1 -28642.114,E2 -28642.114} C_VEL
LIN {X 0,Y 65.791,Z 472.341,A -85,B 0,C 180,E1 -28647.626,E2 -28647.626} C_VEL
LIN {X 0,Y 66.588,Z 462.748,A -85,B 0,C 180,E1 -28652.658,E2 -28652.658} C_VEL
LIN {X 0,Y 67.652,Z 451.828,A -85,B 0,C 180,E1 -28657.148,E2 -28657.148} C_VEL
LIN {X 0,Y 68.789,Z 439.601,A -85,B 0,C 180,E1 -28660.897,E2 -28660.897} C_VEL
LIN {X 0,Y 68.647,Z 433.93,A -85,B 0,C 180,E1 -28662.239,E2 -28662.239} C_VEL
LIN {X 0,Y 66.369,Z 424.489,A -85,B 0,C 180,E1 -28663.992,E2 -28663.992} C_VEL
LIN {X 0,Y 64.015,Z 414.964,A -85,B 0,C 180,E1 -28665.618,E2 -28665.618} C_VEL
LIN {X 0,Y 63.787,Z 409.151,A -85,B 0,C 180,E1 -28666.68,E2 -28666.68} C_VEL
LIN {X 0,Y 65.649,Z 381.948,A -85,B 0,C 180,E1 -28671.655,E2 -28671.655} C_VEL
LIN {X 0,Y 64.109,Z 357.106,A -85,B 0,C 180,E1 -28676.414,E2 -28676.414} C_VEL
LIN {X 0,Y 60.371,Z 342.185,A -85,B 0,C 180,E1 -28680.094,E2 -28680.094} C_VEL
LIN {X 0,Y 59.251,Z 337.176,A -85,B 0,C 180,E1 -28687.313,E2 -28687.313} C_VEL
LIN {X 0,Y 58.484,Z 333.197,A -85,B 0,C 180,E1 -28693.528,E2 -28693.528} C_VEL
LIN {X 0,Y 58.605,Z 333.174,A -85,B 0,C 180,E1 -28696.11,E2 -28696.11} C_VEL
LIN {X 0,Y 58.773,Z 333.158,A -85,B 0,C 180,E1 -28703.119,E2 -28703.119} C_VEL
LIN {X 0,Y 59.337,Z 333.094,A -85,B 0,C 180,E1 -28709.986,E2 -28709.986} C_VEL
LIN {X 0,Y 58.773,Z 333.162,A -85,B 0,C 180,E1 -28716.853,E2 -28716.853} C_VEL
LIN {X 0,Y 58.455,Z 333.202,A -85,B 0,C 180,E1 -28725.868,E2 -28725.868} C_VEL
LIN {X 0,Y 58.155,Z 333.231,A -85,B 0,C 180,E1 -28731.239,E2 -28731.239} C_VEL
LIN {X 0,Y 58.12,Z 333.238,A -85,B 0,C 180,E1 -28738.908,E2 -28738.908} C_VEL
LIN {X 0,Y 58.006,Z 333.255,A -85,B 0,C 180,E1 -28747.264,E2 -28747.264} C_VEL
LIN {X 0,Y 57.986,Z 333.255,A -85,B 0,C 180,E1 -28756.627,E2 -28756.627} C_VEL
LIN {X 0,Y 58.001,Z 333.261,A -85,B 0,C 180,E1 -28762.705,E2 -28762.705} C_VEL
LIN {X 0,Y 58.109,Z 333.246,A -85,B 0,C 180,E1 -28771.063,E2 -28771.063} C_VEL
LIN {X 0,Y 58.138,Z 333.239,A -85,B 0,C 180,E1 -28778.733,E2 -28778.733} C_VEL
LIN {X 0,Y 58.571,Z 333.18,A -85,B 0,C 180,E1 -28786.111,E2 -28786.111} C_VEL
LIN {X 0,Y 58.754,Z 333.157,A -85,B 0,C 180,E1 -28793.126,E2 -28793.126} C_VEL
LIN {X 0,Y 59.32,Z 333.094,A -85,B 0,C 180,E1 -28799.996,E2 -28799.996} C_VEL
LIN {X 0,Y 58.756,Z 333.166,A -85,B 0,C 180,E1 -28806.866,E2 -28806.866} C_VEL
LIN {X 0,Y 58.48,Z 333.201,A -85,B 0,C 180,E1 -28816.036,E2 -28816.036} C_VEL
LIN {X 0,Y 58.122,Z 333.235,A -85,B 0,C 180,E1 -28828.921,E2 -28828.921} C_VEL
LIN {X 0,Y 58.165,Z 333.277,A -85,B 0,C 180,E1 -28832.278,E2 -28832.278} C_VEL
LIN {X 0,Y 59.521,Z 338.779,A -85,B 0,C 180,E1 -28840.493,E2 -28840.493} C_VEL
LIN {X 0,Y 60.542,Z 343.19,A -85,B 0,C 180,E1 -28846.475,E2 -28846.475} C_VEL
LIN {X 0,Y 66.075,Z 365.178,A -85,B 0,C 180,E1 -28851.525,E2 -28851.525} C_VEL
LIN {X 0,Y 66.432,Z 371.61,A -85,B 0,C 180,E1 -28852.69,E2 -28852.69} C_VEL
LIN {X 0,Y 67.008,Z 387.877,A -85,B 0,C 180,E1 -28855.554,E2 -28855.554} C_VEL
LIN {X 0,Y 63.948,Z 438.062,A -85,B 0,C 180,E1 -28864.593,E2 -28864.593} C_VEL
LIN {X 0,Y 63.175,Z 447.77,A -85,B 0,C 180,E1 -28867.101,E2 -28867.101} C_VEL
LIN {X 0,Y 62.319,Z 456.875,A -85,B 0,C 180,E1 -28870.241,E2 -28870.241} C_VEL
LIN {X 0,Y 61.558,Z 466.052,A -85,B 0,C 180,E1 -28874.282,E2 -28874.282} C_VEL
LIN {X 0,Y 60.907,Z 474.935,A -85,B 0,C 180,E1 -28879.207,E2 -28879.207} C_VEL
LIN {X 0,Y 60.637,Z 482.339,A -85,B 0,C 180,E1 -28884.193,E2 -28884.193} C_VEL
LIN {X 0,Y 60.901,Z 489.666,A -85,B 0,C 180,E1 -28890.013,E2 -28890.013} C_VEL
LIN {X 0,Y 61.786,Z 496.693,A -85,B 0,C 180,E1 -28896.544,E2 -28896.544} C_VEL
LIN {X 0,Y 62.114,Z 499.497,A -85,B 0,C 180,E1 -28899.784,E2 -28899.784} C_VEL
LIN {X 0,Y 62.01,Z 504.019,A -85,B 0,C 180,E1 -28906.472,E2 -28906.472} C_VEL
LIN {X 0,Y 63.489,Z 509.735,A -85,B 0,C 180,E1 -28916.293,E2 -28916.293} C_VEL
LIN {X 0,Y 68.408,Z 515.8,A -85,B 0,C 180,E1 -28928.066,E2 -28928.066} C_VEL
LIN {X 0,Y 74.066,Z 519.514,A -85,B 0,C 180,E1 -28935.38,E2 -28935.38} C_VEL
LIN {X 0,Y 80.906,Z 522.479,A -85,B 0,C 180,E1 -28941.434,E2 -28941.434} C_VEL
LIN {X 0,Y 88.329,Z 524.72,A -85,B 0,C 180,E1 -28946.157,E2 -28946.157} C_VEL
LIN {X 0,Y 89.862,Z 524.88,A -85,B 0,C 180,E1 -28948.139,E2 -28948.139} C_VEL
LIN {X 0,Y 79.963,Z 520.585,A -85,B 0,C 180,E1 -28953.934,E2 -28953.934} C_VEL
LIN {X 0,Y 72.545,Z 515.801,A -85,B 0,C 180,E1 -28960.183,E2 -28960.183} C_VEL
LIN {X 0,Y 66.523,Z 509.88,A -85,B 0,C 180,E1 -28967.805,E2 -28967.805} C_VEL
LIN {X 0,Y 62.074,Z 502.746,A -85,B 0,C 180,E1 -28976.758,E2 -28976.758} C_VEL
LIN {X 0,Y 59.768,Z 495.597,A -85,B 0,C 180,E1 -28985.063,E2 -28985.063} C_VEL
LIN {X 0,Y 58.9,Z 488.905,A -85,B 0,C 180,E1 -28992.056,E2 -28992.056} C_VEL
LIN {X 0,Y 58.673,Z 481.392,A -85,B 0,C 180,E1 -28998.802,E2 -28998.802} C_VEL
LIN {X 0,Y 58.907,Z 472.111,A -85,B 0,C 180,E1 -29005.63,E2 -29005.63} C_VEL
LIN {X 0,Y 59.606,Z 462.379,A -85,B 0,C 180,E1 -29011.332,E2 -29011.332} C_VEL
LIN {X 0,Y 60.511,Z 452.159,A -85,B 0,C 180,E1 -29016.018,E2 -29016.018} C_VEL
LIN {X 0,Y 61.697,Z 439.439,A -85,B 0,C 180,E1 -29020.386,E2 -29020.386} C_VEL
LIN {X 0,Y 63.08,Z 420.226,A -85,B 0,C 180,E1 -29024.557,E2 -29024.557} C_VEL
LIN {X 0,Y 63.787,Z 409.151,A -85,B 0,C 180,E1 -29026.68,E2 -29026.68} C_VEL
LIN {X 0,Y 63.682,Z 403.382,A -85,B 0,C 180,E1 -29027.78,E2 -29027.78} C_VEL
LIN {X 0,Y 61.693,Z 393.925,A -85,B 0,C 180,E1 -29029.691,E2 -29029.691} C_VEL
LIN {X 0,Y 58.822,Z 382.566,A -85,B 0,C 180,E1 -29032.19,E2 -29032.19} C_VEL
LIN {X 0,Y 58.321,Z 378.7,A -85,B 0,C 180,E1 -29033.034,E2 -29033.034} C_VEL
LIN {X 0,Y 57.31,Z 358.891,A -85,B 0,C 180,E1 -29037.28,E2 -29037.28} C_VEL
LIN {X 0,Y 53.149,Z 342.366,A -85,B 0,C 180,E1 -29041.881,E2 -29041.881} C_VEL
LIN {X 0,Y 51.849,Z 336.456,A -85,B 0,C 180,E1 -29051.604,E2 -29051.604} C_VEL
LIN {X 0,Y 51.565,Z 334.051,A -85,B 0,C 180,E1 -29056.186,E2 -29056.186} C_VEL
LIN {X 0,Y 52.223,Z 333.98,A -85,B 0,C 180,E1 -29069.984,E2 -29069.984} C_VEL
LIN {X 0,Y 51.649,Z 334.051,A -85,B 0,C 180,E1 -29077.804,E2 -29077.804} C_VEL
LIN {X 0,Y 51.335,Z 334.09,A -85,B 0,C 180,E1 -29086.584,E2 -29086.584} C_VEL
LIN {X 0,Y 50.994,Z 334.129,A -85,B 0,C 180,E1 -29094.402,E2 -29094.402} C_VEL
LIN {X 0,Y 51,Z 334.132,A -85,B 0,C 180,E1 -29104.219,E2 -29104.219} C_VEL
LIN {X 0,Y 50.953,Z 334.132,A -85,B 0,C 180,E1 -29116.391,E2 -29116.391} C_VEL
LIN {X 0,Y 50.994,Z 334.123,A -85,B 0,C 180,E1 -29126.54,E2 -29126.54} C_VEL
LIN {X 0,Y 50.98,Z 334.124,A -85,B 0,C 180,E1 -29135.566,E2 -29135.566} C_VEL
LIN {X 0,Y 51.354,Z 334.078,A -85,B 0,C 180,E1 -29144.111,E2 -29144.111} C_VEL
LIN {X 0,Y 51.629,Z 334.047,A -85,B 0,C 180,E1 -29152.172,E2 -29152.172} C_VEL
LIN {X 0,Y 52.206,Z 333.979,A -85,B 0,C 180,E1 -29159.996,E2 -29159.996} C_VEL
LIN {X 0,Y 51.634,Z 334.053,A -85,B 0,C 180,E1 -29167.819,E2 -29167.819} C_VEL
LIN {X 0,Y 51.339,Z 334.09,A -85,B 0,C 180,E1 -29176.689,E2 -29176.689} C_VEL
LIN {X 0,Y 51.142,Z 334.221,A -85,B 0,C 180,E1 -29189.873,E2 -29189.873} C_VEL
LIN {X 0,Y 52.49,Z 339.899,A -85,B 0,C 180,E1 -29199.722,E2 -29199.722} C_VEL
LIN {X 0,Y 53.197,Z 343.037,A -85,B 0,C 180,E1 -29204.57,E2 -29204.57} C_VEL
LIN {X 0,Y 57.539,Z 359.63,A -85,B 0,C 180,E1 -29209.088,E2 -29209.088} C_VEL
LIN {X 0,Y 59.353,Z 368.408,A -85,B 0,C 180,E1 -29211.151,E2 -29211.151} C_VEL
LIN {X 0,Y 59.96,Z 387.747,A -85,B 0,C 180,E1 -29214.968,E2 -29214.968} C_VEL
LIN {X 0,Y 56.838,Z 438.723,A -85,B 0,C 180,E1 -29225.353,E2 -29225.353} C_VEL
LIN {X 0,Y 56.016,Z 448.635,A -85,B 0,C 180,E1 -29228.392,E2 -29228.392} C_VEL
LIN {X 0,Y 55.199,Z 458.383,A -85,B 0,C 180,E1 -29232.416,E2 -29232.416} C_VEL
LIN {X 0,Y 54.463,Z 468.6,A -85,B 0,C 180,E1 -29237.912,E2 -29237.912} C_VEL
LIN {X 0,Y 54.125,Z 479.399,A -85,B 0,C 180,E1 -29245.361,E2 -29245.361} C_VEL
LIN {X 0,Y 54.737,Z 488.976,A -85,B 0,C 180,E1 -29253.695,E2 -29253.695} C_VEL
LIN {X 0,Y 55.864,Z 495.907,A -85,B 0,C 180,E1 -29260.891,E2 -29260.891} C_VEL
LIN {X 0,Y 55.955,Z 499.584,A -85,B 0,C 180,E1 -29266.429,E2 -29266.429} C_VEL
LIN {X 0,Y 57.814,Z 506.716,A -85,B 0,C 180,E1 -29279.107,E2 -29279.107} C_VEL
LIN {X 0,Y 63.306,Z 513.31,A -85,B 0,C 180,E1 -29291.779,E2 -29291.779} C_VEL
LIN {X 0,Y 71.834,Z 518.406,A -85,B 0,C 180,E1 -29301.519,E2 -29301.519} C_VEL
LIN {X 0,Y 76.834,Z 520.5,A -85,B 0,C 180,E1 -29305.42,E2 -29305.42} C_VEL
LIN {X 0,Y 79.05,Z 521.231,A -85,B 0,C 180,E1 -29307.765,E2 -29307.765} C_VEL
LIN {X 0,Y 70.695,Z 516.462,A -85,B 0,C 180,E1 -29313.486,E2 -29313.486} C_VEL
LIN {X 0,Y 62.547,Z 509.636,A -85,B 0,C 180,E1 -29322.005,E2 -29322.005} C_VEL
LIN {X 0,Y 57.767,Z 503.423,A -85,B 0,C 180,E1 -29329.894,E2 -29329.894} C_VEL
LIN {X 0,Y 54.62,Z 496.832,A -85,B 0,C 180,E1 -29338.161,E2 -29338.161} C_VEL
LIN {X 0,Y 52.748,Z 488.679,A -85,B 0,C 180,E1 -29347.661,E2 -29347.661} C_VEL
LIN {X 0,Y 52.164,Z 480.664,A -85,B 0,C 180,E1 -29355.636,E2 -29355.636} C_VEL
LIN {X 0,Y 52.159,Z 472.214,A -85,B 0,C 180,E1 -29362.637,E2 -29362.637} C_VEL
LIN {X 0,Y 52.613,Z 462.855,A -85,B 0,C 180,E1 -29368.966,E2 -29368.966} C_VEL
LIN {X 0,Y 53.355,Z 452.912,A -85,B 0,C 180,E1 -29374.291,E2 -29374.291} C_VEL
LIN {X 0,Y 54.144,Z 444.185,A -85,B 0,C 180,E1 -29377.955,E2 -29377.955} C_VEL
LIN {X 0,Y 55.151,Z 433.186,A -85,B 0,C 180,E1 -29381.385,E2 -29381.385} C_VEL
LIN {X 0,Y 58.624,Z 383.822,A -85,B 0,C 180,E1 -29391.95,E2 -29391.95} C_VEL
LIN {X 0,Y 58.321,Z 378.7,A -85,B 0,C 180,E1 -29393.034,E2 -29393.034} C_VEL
LIN {X 0,Y 57.295,Z 373.005,A -85,B 0,C 180,E1 -29394.349,E2 -29394.349} C_VEL
LIN {X 0,Y 53.864,Z 363.995,A -85,B 0,C 180,E1 -29396.863,E2 -29396.863} C_VEL
LIN {X 0,Y 50.587,Z 356.919,A -85,B 0,C 180,E1 -29399.149,E2 -29399.149} C_VEL
LIN {X 0,Y 47.9,Z 349.636,A -85,B 0,C 180,E1 -29401.62,E2 -29401.62} C_VEL
LIN {X 0,Y 45.878,Z 342.2,A -85,B 0,C 180,E1 -29404.437,E2 -29404.437} C_VEL
LIN {X 0,Y 44.76,Z 336.137,A -85,B 0,C 180,E1 -29416.369,E2 -29416.369} C_VEL
LIN {X 0,Y 44.499,Z 334.939,A -85,B 0,C 180,E1 -29419.176,E2 -29419.176} C_VEL
LIN {X 0,Y 45.1,Z 334.867,A -85,B 0,C 180,E1 -29429.982,E2 -29429.982} C_VEL
LIN {X 0,Y 44.494,Z 334.942,A -85,B 0,C 180,E1 -29439.069,E2 -29439.069} C_VEL
LIN {X 0,Y 44.103,Z 334.989,A -85,B 0,C 180,E1 -29448.563,E2 -29448.563} C_VEL
LIN {X 0,Y 43.806,Z 335.02,A -85,B 0,C 180,E1 -29458.746,E2 -29458.746} C_VEL
LIN {X 0,Y 43.817,Z 335.023,A -85,B 0,C 180,E1 -29466.672,E2 -29466.672} C_VEL
LIN {X 0,Y 43.765,Z 335.025,A -85,B 0,C 180,E1 -29480.027,E2 -29480.027} C_VEL
LIN {X 0,Y 43.795,Z 335.029,A -85,B 0,C 180,E1 -29491.216,E2 -29491.216} C_VEL
LIN {X 0,Y 44.162,Z 334.978,A -85,B 0,C 180,E1 -29502.634,E2 -29502.634} C_VEL
LIN {X 0,Y 44.47,Z 334.943,A -85,B 0,C 180,E1 -29510.902,E2 -29510.902} C_VEL
LIN {X 0,Y 45.082,Z 334.866,A -85,B 0,C 180,E1 -29519.995,E2 -29519.995} C_VEL
LIN {X 0,Y 44.494,Z 334.938,A -85,B 0,C 180,E1 -29529.083,E2 -29529.083} C_VEL
LIN {X 0,Y 44.119,Z 334.982,A -85,B 0,C 180,E1 -29538.573,E2 -29538.573} C_VEL
LIN {X 0,Y 43.99,Z 335.108,A -85,B 0,C 180,E1 -29546.696,E2 -29546.696} C_VEL
LIN {X 0,Y 45.086,Z 339.532,A -85,B 0,C 180,E1 -29555.765,E2 -29555.765} C_VEL
LIN {X 0,Y 45.894,Z 342.917,A -85,B 0,C 180,E1 -29562.194,E2 -29562.194} C_VEL
LIN {X 0,Y 50.334,Z 359.705,A -85,B 0,C 180,E1 -29567.642,E2 -29567.642} C_VEL
LIN {X 0,Y 52.351,Z 369.081,A -85,B 0,C 180,E1 -29570.157,E2 -29570.157} C_VEL
LIN {X 0,Y 52.852,Z 388.408,A -85,B 0,C 180,E1 -29574.497,E2 -29574.497} C_VEL
LIN {X 0,Y 49.854,Z 437.738,A -85,B 0,C 180,E1 -29586.111,E2 -29586.111} C_VEL
LIN {X 0,Y 49.059,Z 447.735,A -85,B 0,C 180,E1 -29589.582,E2 -29589.582} C_VEL
LIN {X 0,Y 48.335,Z 457.582,A -85,B 0,C 180,E1 -29594.198,E2 -29594.198} C_VEL
LIN {X 0,Y 47.753,Z 467.825,A -85,B 0,C 180,E1 -29600.488,E2 -29600.488} C_VEL
LIN {X 0,Y 47.698,Z 478.611,A -85,B 0,C 180,E1 -29608.962,E2 -29608.962} C_VEL
LIN {X 0,Y 48.792,Z 488.237,A -85,B 0,C 180,E1 -29618.298,E2 -29618.298} C_VEL
LIN {X 0,Y 49.968,Z 493.389,A -85,B 0,C 180,E1 -29624.264,E2 -29624.264} C_VEL
LIN {X 0,Y 50.683,Z 499.334,A -85,B 0,C 180,E1 -29634.597,E2 -29634.597} C_VEL
LIN {X 0,Y 54.228,Z 506.268,A -85,B 0,C 180,E1 -29647.922,E2 -29647.922} C_VEL
LIN {X 0,Y 62.963,Z 513.406,A -85,B 0,C 180,E1 -29661.398,E2 -29661.398} C_VEL
LIN {X 0,Y 67.872,Z 516.027,A -85,B 0,C 180,E1 -29665.946,E2 -29665.946} C_VEL
LIN {X 0,Y 68.267,Z 516.064,A -85,B 0,C 180,E1 -29667.608,E2 -29667.608} C_VEL
LIN {X 0,Y 59.307,Z 509.23,A -85,B 0,C 180,E1 -29675.5,E2 -29675.5} C_VEL
LIN {X 0,Y 53.873,Z 503.349,A -85,B 0,C 180,E1 -29682.935,E2 -29682.935} C_VEL
LIN {X 0,Y 49.704,Z 496.405,A -85,B 0,C 180,E1 -29691.876,E2 -29691.876} C_VEL
LIN {X 0,Y 47.041,Z 488.252,A -85,B 0,C 180,E1 -29702.145,E2 -29702.145} C_VEL
LIN {X 0,Y 45.925,Z 480.42,A -85,B 0,C 180,E1 -29711.033,E2 -29711.033} C_VEL
LIN {X 0,Y 45.562,Z 473.211,A -85,B 0,C 180,E1 -29717.974,E2 -29717.974} C_VEL
LIN {X 0,Y 45.677,Z 464.656,A -85,B 0,C 180,E1 -29724.848,E2 -29724.848} C_VEL
LIN {X 0,Y 46.222,Z 455.413,A -85,B 0,C 180,E1 -29730.88,E2 -29730.88} C_VEL
LIN {X 0,Y 47.053,Z 445.263,A -85,B 0,C 180,E1 -29736.029,E2 -29736.029} C_VEL
LIN {X 0,Y 47.965,Z 434.412,A -85,B 0,C 180,E1 -29740.075,E2 -29740.075} C_VEL
LIN {X 0,Y 50.46,Z 396.323,A -85,B 0,C 180,E1 -29749.812,E2 -29749.812} C_VEL
LIN {X 0,Y 51.529,Z 382.319,A -85,B 0,C 180,E1 -29753.055,E2 -29753.055} C_VEL
LIN {X 0,Y 50.226,Z 359.39,A -85,B 0,C 180,E1 -29758.631,E2 -29758.631} C_VEL
LIN {X 0,Y 47.9,Z 349.636,A -85,B 0,C 180,E1 -29761.62,E2 -29761.62} C_VEL
LIN {X 0,Y 46.305,Z 346.285,A -85,B 0,C 180,E1 -29763.303,E2 -29763.303} C_VEL
LIN {X 0,Y 44.026,Z 343.609,A -85,B 0,C 180,E1 -29765.79,E2 -29765.79} C_VEL
LIN {X 0,Y 40.795,Z 340.785,A -85,B 0,C 180,E1 -29770.425,E2 -29770.425} C_VEL
LIN {X 0,Y 38.31,Z 338.259,A -85,B 0,C 180,E1 -29776.648,E2 -29776.648} C_VEL
LIN {X 0,Y 37.715,Z 336.928,A -85,B 0,C 180,E1 -29780.203,E2 -29780.203} C_VEL
LIN {X 0,Y 37.537,Z 335.8,A -85,B 0,C 180,E1 -29783.259,E2 -29783.259} C_VEL
LIN {X 0,Y 37.959,Z 335.756,A -85,B 0,C 180,E1 -29789.979,E2 -29789.979} C_VEL
LIN {X 0,Y 37.274,Z 335.834,A -85,B 0,C 180,E1 -29800.845,E2 -29800.845} C_VEL
LIN {X 0,Y 37.026,Z 335.87,A -85,B 0,C 180,E1 -29808.35,E2 -29808.35} C_VEL
LIN {X 0,Y 36.697,Z 335.914,A -85,B 0,C 180,E1 -29825.037,E2 -29825.037} C_VEL
LIN {X 0,Y 36.701,Z 335.902,A -85,B 0,C 180,E1 -29829.997,E2 -29829.997} C_VEL
LIN {X 0,Y 36.691,Z 335.905,A -85,B 0,C 180,E1 -29839.971,E2 -29839.971} C_VEL
LIN {X 0,Y 36.678,Z 335.909,A -85,B 0,C 180,E1 -29844.904,E2 -29844.904} C_VEL
LIN {X 0,Y 37.011,Z 335.872,A -85,B 0,C 180,E1 -29861.615,E2 -29861.615} C_VEL
LIN {X 0,Y 37.269,Z 335.843,A -85,B 0,C 180,E1 -29869.124,E2 -29869.124} C_VEL
LIN {X 0,Y 37.94,Z 335.754,A -85,B 0,C 180,E1 -29879.994,E2 -29879.994} C_VEL
LIN {X 0,Y 37.294,Z 335.829,A -85,B 0,C 180,E1 -29890.856,E2 -29890.856} C_VEL
LIN {X 0,Y 36.957,Z 336.012,A -85,B 0,C 180,E1 -29902.348,E2 -29902.348} C_VEL
LIN {X 0,Y 38.021,Z 340.453,A -85,B 0,C 180,E1 -29913.672,E2 -29913.672} C_VEL
LIN {X 0,Y 38.644,Z 342.854,A -85,B 0,C 180,E1 -29919.106,E2 -29919.106} C_VEL
LIN {X 0,Y 42.546,Z 357.386,A -85,B 0,C 180,E1 -29925.001,E2 -29925.001} C_VEL
LIN {X 0,Y 45.323,Z 369.95,A -85,B 0,C 180,E1 -29929.1,E2 -29929.1} C_VEL
LIN {X 0,Y 45.753,Z 388.434,A -85,B 0,C 180,E1 -29933.916,E2 -29933.916} C_VEL
LIN {X 0,Y 42.837,Z 437.556,A -85,B 0,C 180,E1 -29947.409,E2 -29947.409} C_VEL
LIN {X 0,Y 42.137,Z 446.838,A -85,B 0,C 180,E1 -29951.169,E2 -29951.169} C_VEL
LIN {X 0,Y 41.522,Z 456.761,A -85,B 0,C 180,E1 -29956.564,E2 -29956.564} C_VEL
LIN {X 0,Y 41.183,Z 465.458,A -85,B 0,C 180,E1 -29962.667,E2 -29962.667} C_VEL
LIN {X 0,Y 41.361,Z 473.958,A -85,B 0,C 180,E1 -29970.02,E2 -29970.02} C_VEL
LIN {X 0,Y 42.26,Z 482.132,A -85,B 0,C 180,E1 -29978.386,E2 -29978.386} C_VEL
LIN {X 0,Y 43.993,Z 489.324,A -85,B 0,C 180,E1 -29986.661,E2 -29986.661} C_VEL
LIN {X 0,Y 44.521,Z 492.03,A -85,B 0,C 180,E1 -29990.822,E2 -29990.822} C_VEL
LIN {X 0,Y 47.253,Z 500.098,A -85,B 0,C 180,E1 -30006.524,E2 -30006.524} C_VEL
LIN {X 0,Y 54.364,Z 507.465,A -85,B 0,C 180,E1 -30020.882,E2 -30020.882} C_VEL
LIN {X 0,Y 59.123,Z 510.592,A -85,B 0,C 180,E1 -30026.331,E2 -30026.331} C_VEL
LIN {X 0,Y 51.842,Z 504.094,A -85,B 0,C 180,E1 -30033.863,E2 -30033.863} C_VEL
LIN {X 0,Y 46.43,Z 497.377,A -85,B 0,C 180,E1 -30042.383,E2 -30042.383} C_VEL
LIN {X 0,Y 42.553,Z 489.85,A -85,B 0,C 180,E1 -30052.384,E2 -30052.384} C_VEL
LIN {X 0,Y 40.453,Z 482.047,A -85,B 0,C 180,E1 -30062.495,E2 -30062.495} C_VEL
LIN {X 0,Y 39.418,Z 474.127,A -85,B 0,C 180,E1 -30071.576,E2 -30071.576} C_VEL
LIN {X 0,Y 39.096,Z 464.199,A -85,B 0,C 180,E1 -30081.077,E2 -30081.077} C_VEL
LIN {X 0,Y 39.393,Z 455.293,A -85,B 0,C 180,E1 -30087.972,E2 -30087.972} C_VEL
LIN {X 0,Y 40.058,Z 445.155,A -85,B 0,C 180,E1 -30094.009,E2 -30094.009} C_VEL
LIN {X 0,Y 40.952,Z 434.009,A -85,B 0,C 180,E1 -30098.871,E2 -30098.871} C_VEL
LIN {X 0,Y 43.371,Z 396.618,A -85,B 0,C 180,E1 -30110.029,E2 -30110.029} C_VEL
LIN {X 0,Y 44.443,Z 382.324,A -85,B 0,C 180,E1 -30113.863,E2 -30113.863} C_VEL
LIN {X 0,Y 43.273,Z 360.437,A -85,B 0,C 180,E1 -30120.087,E2 -30120.087} C_VEL
LIN {X 0,Y 39.7,Z 345.977,A -85,B 0,C 180,E1 -30125.659,E2 -30125.659} C_VEL
LIN {X 0,Y 38.556,Z 342.199,A -85,B 0,C 180,E1 -30127.731,E2 -30127.731} C_VEL
LIN {X 0,Y 37.799,Z 337.288,A -85,B 0,C 180,E1 -30139.264,E2 -30139.264} C_VEL
LIN {X 0,Y 37.715,Z 336.928,A -85,B 0,C 180,E1 -30140.203,E2 -30140.203} C_VEL
LIN {X 0,Y 36.876,Z 336.061,A -85,B 0,C 180,E1 -30144.573,E2 -30144.573} C_VEL
LIN {X 0,Y 34.838,Z 336.14,A -85,B 0,C 180,E1 -30151.067,E2 -30151.067} C_VEL
LIN {X 0,Y 29.543,Z 336.66,A -85,B 0,C 180,E1 -30174.471,E2 -30174.471} C_VEL
LIN {X 0,Y 29.468,Z 336.675,A -85,B 0,C 180,E1 -30178.455,E2 -30178.455} C_VEL
LIN {X 0,Y 29.521,Z 336.67,A -85,B 0,C 180,E1 -30195.533,E2 -30195.533} C_VEL
LIN {X 0,Y 29.452,Z 336.678,A -85,B 0,C 180,E1 -30211.486,E2 -30211.486} C_VEL
LIN {X 0,Y 29.821,Z 336.643,A -85,B 0,C 180,E1 -30220.41,E2 -30220.41} C_VEL
LIN {X 0,Y 30.055,Z 336.619,A -85,B 0,C 180,E1 -30226.47,E2 -30226.47} C_VEL
LIN {X 0,Y 30.757,Z 336.555,A -85,B 0,C 180,E1 -30239.993,E2 -30239.993} C_VEL
LIN {X 0,Y 30.022,Z 336.731,A -85,B 0,C 180,E1 -30255.451,E2 -30255.451} C_VEL
LIN {X 0,Y 30.994,Z 341.443,A -85,B 0,C 180,E1 -30270.669,E2 -30270.669} C_VEL
LIN {X 0,Y 31.3,Z 342.811,A -85,B 0,C 180,E1 -30274.628,E2 -30274.628} C_VEL
LIN {X 0,Y 34.309,Z 353.117,A -85,B 0,C 180,E1 -30280.437,E2 -30280.437} C_VEL
LIN {X 0,Y 38.205,Z 369.895,A -85,B 0,C 180,E1 -30287.369,E2 -30287.369} C_VEL
LIN {X 0,Y 38.671,Z 388.642,A -85,B 0,C 180,E1 -30293.188,E2 -30293.188} C_VEL
LIN {X 0,Y 35.869,Z 437.018,A -85,B 0,C 180,E1 -30309.225,E2 -30309.225} C_VEL
LIN {X 0,Y 35.271,Z 446.867,A -85,B 0,C 180,E1 -30314.124,E2 -30314.124} C_VEL
LIN {X 0,Y 34.891,Z 455.585,A -85,B 0,C 180,E1 -30319.873,E2 -30319.873} C_VEL
LIN {X 0,Y 34.846,Z 464.332,A -85,B 0,C 180,E1 -30327.133,E2 -30327.133} C_VEL
LIN {X 0,Y 35.557,Z 474.111,A -85,B 0,C 180,E1 -30337.114,E2 -30337.114} C_VEL
LIN {X 0,Y 37.223,Z 482.171,A -85,B 0,C 180,E1 -30346.473,E2 -30346.473} C_VEL
LIN {X 0,Y 38.463,Z 486.234,A -85,B 0,C 180,E1 -30351.455,E2 -30351.455} C_VEL
LIN {X 0,Y 39.063,Z 488.003,A -85,B 0,C 180,E1 -30354.045,E2 -30354.045} C_VEL
LIN {X 0,Y 41.82,Z 495.272,A -85,B 0,C 180,E1 -30369.085,E2 -30369.085} C_VEL
LIN {X 0,Y 48.373,Z 502.451,A -85,B 0,C 180,E1 -30383.334,E2 -30383.334} C_VEL
LIN {X 0,Y 49.809,Z 503.555,A -85,B 0,C 180,E1 -30385.645,E2 -30385.645} C_VEL
LIN {X 0,Y 43.443,Z 496.721,A -85,B 0,C 180,E1 -30393.59,E2 -30393.59} C_VEL
LIN {X 0,Y 38.202,Z 488.626,A -85,B 0,C 180,E1 -30404.264,E2 -30404.264} C_VEL
LIN {X 0,Y 35.292,Z 481.081,A -85,B 0,C 180,E1 -30414.865,E2 -30414.865} C_VEL
LIN {X 0,Y 33.739,Z 473.656,A -85,B 0,C 180,E1 -30424.487,E2 -30424.487} C_VEL
LIN {X 0,Y 32.897,Z 465.346,A -85,B 0,C 180,E1 -30433.913,E2 -30433.913} C_VEL
LIN {X 0,Y 32.752,Z 454.84,A -85,B 0,C 180,E1 -30443.732,E2 -30443.732} C_VEL
LIN {X 0,Y 33.219,Z 444.787,A -85,B 0,C 180,E1 -30451.077,E2 -30451.077} C_VEL
LIN {X 0,Y 34.105,Z 431.926,A -85,B 0,C 180,E1 -30457.812,E2 -30457.812} C_VEL
LIN {X 0,Y 37.403,Z 382.723,A -85,B 0,C 180,E1 -30474.843,E2 -30474.843} C_VEL
LIN {X 0,Y 36.36,Z 361.574,A -85,B 0,C 180,E1 -30481.995,E2 -30481.995} C_VEL
LIN {X 0,Y 32.996,Z 347.584,A -85,B 0,C 180,E1 -30488.501,E2 -30488.501} C_VEL
LIN {X 0,Y 31.34,Z 342.302,A -85,B 0,C 180,E1 -30492.015,E2 -30492.015} C_VEL
LIN {X 0,Y 30.905,Z 338.446,A -85,B 0,C 180,E1 -30503.445,E2 -30503.445} C_VEL
LIN {X 0,Y 30.774,Z 336.555,A -85,B 0,C 180,E1 -30509.974,E2 -30509.974} C_VEL
LIN {X 0,Y 30.066,Z 336.617,A -85,B 0,C 180,E1 -30523.489,E2 -30523.489} C_VEL
LIN {X 0,Y 29.543,Z 336.66,A -85,B 0,C 180,E1 -30534.471,E2 -30534.471} C_VEL
LIN {X 0,Y 28.838,Z 336.735,A -85,B 0,C 180,E1 -30540.623,E2 -30540.623} C_VEL
LIN {X 0,Y 26.894,Z 336.913,A -85,B 0,C 180,E1 -30549.178,E2 -30549.178} C_VEL
LIN {X 0,Y 22.541,Z 337.074,A -85,B 0,C 180,E1 -30576.764,E2 -30576.764} C_VEL
LIN {X 0,Y 22.648,Z 337.07,A -85,B 0,C 180,E1 -30580.315,E2 -30580.315} C_VEL
LIN {X 0,Y 23.445,Z 337.046,A -85,B 0,C 180,E1 -30601.064,E2 -30601.064} C_VEL
LIN {X 0,Y 23.608,Z 340.238,A -85,B 0,C 180,E1 -30617.31,E2 -30617.31} C_VEL
LIN {X 0,Y 24.078,Z 342.966,A -85,B 0,C 180,E1 -30627.988,E2 -30627.988} C_VEL
LIN {X 0,Y 26.521,Z 350.408,A -85,B 0,C 180,E1 -30634.262,E2 -30634.262} C_VEL
LIN {X 0,Y 30.147,Z 365.737,A -85,B 0,C 180,E1 -30643.21,E2 -30643.21} C_VEL
LIN {X 0,Y 31.376,Z 372.357,A -85,B 0,C 180,E1 -30646.246,E2 -30646.246} C_VEL
LIN {X 0,Y 31.591,Z 388.389,A -85,B 0,C 180,E1 -30652.318,E2 -30652.318} C_VEL
LIN {X 0,Y 28.99,Z 436.869,A -85,B 0,C 180,E1 -30672.391,E2 -30672.391} C_VEL
LIN {X 0,Y 28.521,Z 446.914,A -85,B 0,C 180,E1 -30678.748,E2 -30678.748} C_VEL
LIN {X 0,Y 28.479,Z 456.201,A -85,B 0,C 180,E1 -30686.488,E2 -30686.488} C_VEL
LIN {X 0,Y 28.882,Z 464.192,A -85,B 0,C 180,E1 -30694.685,E2 -30694.685} C_VEL
LIN {X 0,Y 30.213,Z 473.033,A -85,B 0,C 180,E1 -30705.197,E2 -30705.197} C_VEL
LIN {X 0,Y 32.686,Z 481.035,A -85,B 0,C 180,E1 -30715.494,E2 -30715.494} C_VEL
LIN {X 0,Y 34.351,Z 485.043,A -85,B 0,C 180,E1 -30721.139,E2 -30721.139} C_VEL
LIN {X 0,Y 40.242,Z 494.689,A -85,B 0,C 180,E1 -30741.829,E2 -30741.829} C_VEL
LIN {X 0,Y 41.307,Z 495.724,A -85,B 0,C 180,E1 -30743.942,E2 -30743.942} C_VEL
LIN {X 0,Y 35.333,Z 488.063,A -85,B 0,C 180,E1 -30753.421,E2 -30753.421} C_VEL
LIN {X 0,Y 30.139,Z 477.686,A -85,B 0,C 180,E1 -30768.216,E2 -30768.216} C_VEL
LIN {X 0,Y 27.551,Z 467.844,A -85,B 0,C 180,E1 -30781.835,E2 -30781.835} C_VEL
LIN {X 0,Y 26.45,Z 456.271,A -85,B 0,C 180,E1 -30795.418,E2 -30795.418} C_VEL
LIN {X 0,Y 26.475,Z 445.464,A -85,B 0,C 180,E1 -30805.563,E2 -30805.563} C_VEL
LIN {X 0,Y 27.067,Z 433.331,A -85,B 0,C 180,E1 -30813.835,E2 -30813.835} C_VEL
LIN {X 0,Y 29.42,Z 393.276,A -85,B 0,C 180,E1 -30831.971,E2 -30831.971} C_VEL
LIN {X 0,Y 30.295,Z 382.457,A -85,B 0,C 180,E1 -30836.228,E2 -30836.228} C_VEL
LIN {X 0,Y 29.505,Z 362.893,A -85,B 0,C 180,E1 -30844.395,E2 -30844.395} C_VEL
LIN {X 0,Y 26.558,Z 349.929,A -85,B 0,C 180,E1 -30852.153,E2 -30852.153} C_VEL
LIN {X 0,Y 24.369,Z 342.415,A -85,B 0,C 180,E1 -30858.531,E2 -30858.531} C_VEL
LIN {X 0,Y 24.167,Z 339.533,A -85,B 0,C 180,E1 -30869.966,E2 -30869.966} C_VEL
LIN {X 0,Y 22.837,Z 337.064,A -85,B 0,C 180,E1 -30885.583,E2 -30885.583} C_VEL
LIN {X 0,Y 22.535,Z 337.073,A -85,B 0,C 180,E1 -30891.646,E2 -30891.646} C_VEL
LIN {X 0,Y 22.175,Z 337.084,A -85,B 0,C 180,E1 -30909.283,E2 -30909.283} C_VEL
LIN {X 0,Y 22.17,Z 337.085,A -85,B 0,C 180,E1 -30920.64,E2 -30920.64} C_VEL
LIN {X 0,Y 22.648,Z 337.07,A -85,B 0,C 180,E1 -30940.315,E2 -30940.315} C_VEL
LIN {X 0,Y 22.645,Z 337.448,A -85,B 0,C 180,E1 -30946.767,E2 -30946.767} C_VEL
LIN {X 0,Y 22.159,Z 338.375,A -85,B 0,C 180,E1 -30952.944,E2 -30952.944} C_VEL
LIN {X 0,Y 21.033,Z 340.452,A -85,B 0,C 180,E1 -30961.975,E2 -30961.975} C_VEL
LIN {X 0,Y 19.562,Z 344.264,A -85,B 0,C 180,E1 -30973.974,E2 -30973.974} C_VEL
LIN {X 0,Y 19.263,Z 348.371,A -85,B 0,C 180,E1 -30983.28,E2 -30983.28} C_VEL
LIN {X 0,Y 19.613,Z 350.336,A -85,B 0,C 180,E1 -30986.065,E2 -30986.065} C_VEL
LIN {X 0,Y 22.435,Z 362.783,A -85,B 0,C 180,E1 -30997.023,E2 -30997.023} C_VEL
LIN {X 0,Y 24.404,Z 373.006,A -85,B 0,C 180,E1 -31003.67,E2 -31003.67} C_VEL
LIN {X 0,Y 24.531,Z 388.282,A -85,B 0,C 180,E1 -31011.141,E2 -31011.141} C_VEL
LIN {X 0,Y 22.23,Z 436.831,A -85,B 0,C 180,E1 -31037.612,E2 -31037.612} C_VEL
LIN {X 0,Y 22.095,Z 445.52,A -85,B 0,C 180,E1 -31044.733,E2 -31044.733} C_VEL
LIN {X 0,Y 22.595,Z 456.009,A -85,B 0,C 180,E1 -31055.992,E2 -31055.992} C_VEL
LIN {X 0,Y 23.916,Z 464.79,A -85,B 0,C 180,E1 -31067.123,E2 -31067.123} C_VEL
LIN {X 0,Y 26.251,Z 472.908,A -85,B 0,C 180,E1 -31078.012,E2 -31078.012} C_VEL
LIN {X 0,Y 29.373,Z 479.938,A -85,B 0,C 180,E1 -31087.211,E2 -31087.211} C_VEL
LIN {X 0,Y 30.389,Z 481.806,A -85,B 0,C 180,E1 -31090.013,E2 -31090.013} C_VEL
LIN {X 0,Y 33.109,Z 486.461,A -85,B 0,C 180,E1 -31100.455,E2 -31100.455} C_VEL
LIN {X 0,Y 32.376,Z 485.555,A -85,B 0,C 180,E1 -31103.356,E2 -31103.356} C_VEL
LIN {X 0,Y 26.473,Z 475.686,A -85,B 0,C 180,E1 -31116.542,E2 -31116.542} C_VEL
LIN {X 0,Y 23.064,Z 466.695,A -85,B 0,C 180,E1 -31129.451,E2 -31129.451} C_VEL
LIN {X 0,Y 21.108,Z 457.791,A -85,B 0,C 180,E1 -31141.94,E2 -31141.94} C_VEL
LIN {X 0,Y 20.134,Z 446.341,A -85,B 0,C 180,E1 -31156.097,E2 -31156.097} C_VEL
LIN {X 0,Y 20.109,Z 436.958,A -85,B 0,C 180,E1 -31165.222,E2 -31165.222} C_VEL
LIN {X 0,Y 20.405,Z 426.982,A -85,B 0,C 180,E1 -31172.571,E2 -31172.571} C_VEL
LIN {X 0,Y 23.282,Z 383.211,A -85,B 0,C 180,E1 -31197.711,E2 -31197.711} C_VEL
LIN {X 0,Y 22.62,Z 363.477,A -85,B 0,C 180,E1 -31208.585,E2 -31208.585} C_VEL
LIN {X 0,Y 20.071,Z 351.525,A -85,B 0,C 180,E1 -31218.6,E2 -31218.6} C_VEL
LIN {X 0,Y 17.898,Z 343.691,A -85,B 0,C 180,E1 -31228.548,E2 -31228.548} C_VEL
LIN {X 0,Y 17.559,Z 342.399,A -85,B 0,C 180,E1 -31231.387,E2 -31231.387} C_VEL
LIN {X 0,Y 16.82,Z 341.108,A -85,B 0,C 180,E1 -31242.008,E2 -31242.008} C_VEL
LIN {X 0,Y 15.748,Z 340.105,A -85,B 0,C 180,E1 -31256.77,E2 -31256.77} C_VEL
LIN {X 0,Y 15.513,Z 339.396,A -85,B 0,C 180,E1 -31294.83,E2 -31294.83} C_VEL
LIN {X 0,Y 16.983,Z 340.535,A -85,B 0,C 180,E1 -31319.987,E2 -31319.987} C_VEL
LIN {X 0,Y 17.062,Z 342.909,A -85,B 0,C 180,E1 -31334.905,E2 -31334.905} C_VEL
LIN {X 0,Y 19.348,Z 349.356,A -85,B 0,C 180,E1 -31344.937,E2 -31344.937} C_VEL
LIN {X 0,Y 19.613,Z 350.336,A -85,B 0,C 180,E1 -31346.065,E2 -31346.065} C_VEL
LIN {X 0,Y 20.356,Z 355.972,A -85,B 0,C 180,E1 -31350.829,E2 -31350.829} C_VEL
LIN {X 0,Y 20.064,Z 361.827,A -85,B 0,C 180,E1 -31354.126,E2 -31354.126} C_VEL
LIN {X 0,Y 17.594,Z 377.584,A -85,B 0,C 180,E1 -31362.045,E2 -31362.045} C_VEL
LIN {X 0,Y 17.429,Z 381.544,A -85,B 0,C 180,E1 -31364.653,E2 -31364.653} C_VEL
LIN {X 0,Y 17.451,Z 388.273,A -85,B 0,C 180,E1 -31369.285,E2 -31369.285} C_VEL
LIN {X 0,Y 15.909,Z 435.764,A -85,B 0,C 180,E1 -31406.791,E2 -31406.791} C_VEL
LIN {X 0,Y 16.352,Z 445.456,A -85,B 0,C 180,E1 -31417.768,E2 -31417.768} C_VEL
LIN {X 0,Y 17.692,Z 454.916,A -85,B 0,C 180,E1 -31430.387,E2 -31430.387} C_VEL
LIN {X 0,Y 19.904,Z 463.26,A -85,B 0,C 180,E1 -31442.025,E2 -31442.025} C_VEL
LIN {X 0,Y 23.039,Z 470.943,A -85,B 0,C 180,E1 -31452.068,E2 -31452.068} C_VEL
LIN {X 0,Y 24.843,Z 474.31,A -85,B 0,C 180,E1 -31456.091,E2 -31456.091} C_VEL
LIN {X 0,Y 25.098,Z 474.977,A -85,B 0,C 180,E1 -31460.32,E2 -31460.32} C_VEL
LIN {X 0,Y 20.945,Z 467.488,A -85,B 0,C 180,E1 -31469.793,E2 -31469.793} C_VEL
LIN {X 0,Y 17.284,Z 457.842,A -85,B 0,C 180,E1 -31483.062,E2 -31483.062} C_VEL
LIN {X 0,Y 15.061,Z 447.926,A -85,B 0,C 180,E1 -31497.356,E2 -31497.356} C_VEL
LIN {X 0,Y 14.108,Z 437.57,A -85,B 0,C 180,E1 -31511.49,E2 -31511.49} C_VEL
LIN {X 0,Y 13.848,Z 425.693,A -85,B 0,C 180,E1 -31524.32,E2 -31524.32} C_VEL
LIN {X 0,Y 16.256,Z 383.282,A -85,B 0,C 180,E1 -31560.882,E2 -31560.882} C_VEL
LIN {X 0,Y 16.064,Z 365.157,A -85,B 0,C 180,E1 -31574.893,E2 -31574.893} C_VEL
LIN {X 0,Y 14.06,Z 353.401,A -85,B 0,C 180,E1 -31590.056,E2 -31590.056} C_VEL
LIN {X 0,Y 12.928,Z 347.287,A -85,B 0,C 180,E1 -31602.119,E2 -31602.119} C_VEL
LIN {X 0,Y 11.261,Z 345.72,A -85,B 0,C 180,E1 -31617.085,E2 -31617.085} C_VEL
LIN {X 0,Y 10.42,Z 344.876,A -85,B 0,C 180,E1 -31649.655,E2 -31649.655} C_VEL
LIN {X 0,Y 11.127,Z 345.253,A -85,B 0,C 180,E1 -31666.363,E2 -31666.363} C_VEL
LIN {X 0,Y 12.031,Z 346.149,A -85,B 0,C 180,E1 -31676.861,E2 -31676.861} C_VEL
LIN {X 0,Y 12.832,Z 348.841,A -85,B 0,C 180,E1 -31685.877,E2 -31685.877} C_VEL
LIN {X 0,Y 14.086,Z 354.279,A -85,B 0,C 180,E1 -31697.216,E2 -31697.216} C_VEL
LIN {X 0,Y 16.749,Z 369.116,A -85,B 0,C 180,E1 -31715.259,E2 -31715.259} C_VEL
LIN {X 0,Y 17.514,Z 374.135,A -85,B 0,C 180,E1 -31719.619,E2 -31719.619} C_VEL
LIN {X 0,Y 17.429,Z 381.544,A -85,B 0,C 180,E1 -31724.653,E2 -31724.653} C_VEL
LIN {X 0,Y 17.085,Z 385.387,A -85,B 0,C 180,E1 -31727.139,E2 -31727.139} C_VEL
LIN {X 0,Y 16.117,Z 389.148,A -85,B 0,C 180,E1 -31729.499,E2 -31729.499} C_VEL
LIN {X 0,Y 9.692,Z 405.554,A -85,B 0,C 180,E1 -31746.822,E2 -31746.822} C_VEL
LIN {X 0,Y 9.037,Z 411.297,A -85,B 0,C 180,E1 -31755.789,E2 -31755.789} C_VEL
LIN {X 0,Y 10.727,Z 436.472,A -85,B 0,C 180,E1 -31789.2,E2 -31789.2} C_VEL
LIN {X 0,Y 12.599,Z 446.916,A -85,B 0,C 180,E1 -31803.978,E2 -31803.978} C_VEL
LIN {X 0,Y 14.666,Z 453.94,A -85,B 0,C 180,E1 -31813.095,E2 -31813.095} C_VEL
LIN {X 0,Y 14.969,Z 455.183,A -85,B 0,C 180,E1 -31820.557,E2 -31820.557} C_VEL
LIN {X 0,Y 11.732,Z 445.904,A -85,B 0,C 180,E1 -31831.397,E2 -31831.397} C_VEL
LIN {X 0,Y 9.56,Z 436.148,A -85,B 0,C 180,E1 -31845.158,E2 -31845.158} C_VEL
LIN {X 0,Y 8.156,Z 425.036,A -85,B 0,C 180,E1 -31861.554,E2 -31861.554} C_VEL
LIN {X 0,Y 9.292,Z 383.286,A -85,B 0,C 180,E1 -31927.598,E2 -31927.598} C_VEL
LIN {X 0,Y 9.781,Z 366.255,A -85,B 0,C 180,E1 -31949.917,E2 -31949.917} C_VEL
LIN {X 0,Y 9.268,Z 355.907,A -85,B 0,C 180,E1 -31973.274,E2 -31973.274} C_VEL
LIN {X 0,Y 9.301,Z 352.468,A -85,B 0,C 180,E1 -31983.457,E2 -31983.457} C_VEL
LIN {X 0,Y 9.182,Z 351.944,A -85,B 0,C 180,E1 -32017.615,E2 -32017.615} C_VEL
LIN {X 0,Y 9.214,Z 357.324,A -85,B 0,C 180,E1 -32035.901,E2 -32035.901} C_VEL
LIN {X 0,Y 10.34,Z 371.096,A -85,B 0,C 180,E1 -32065.115,E2 -32065.115} C_VEL
LIN {X 0,Y 10.716,Z 375.581,A -85,B 0,C 180,E1 -32071.659,E2 -32071.659} C_VEL
LIN {X 0,Y 10.357,Z 388.411,A -85,B 0,C 180,E1 -32086.091,E2 -32086.091} C_VEL
LIN {X 0,Y 9.037,Z 411.297,A -85,B 0,C 180,E1 -32115.789,E2 -32115.789} C_VEL
LIN {X 0,Y 8.079,Z 411.261,A -85,B 0,C 180,E1 -32118.455,E2 -32118.455} C_VEL
LIN {X 0,Y 6.699,Z 409.986,A -85,B 0,C 180,E1 -32121.313,E2 -32121.313} C_VEL
LIN {X 0,Y 4.136,Z 405.9,A -85,B 0,C 180,E1 -32126.372,E2 -32126.372} C_VEL
LIN {X 0,Y 0.679,Z 393.479,A -85,B 0,C 180,E1 -32303.271,E2 -32303.271} C_VEL
LIN {X 0,Y 2.786,Z 385.057,A -85,B 0,C 180,E1 -32321.611,E2 -32321.611} C_VEL
LIN {X 0,Y 3.233,Z 382.221,A -85,B 0,C 180,E1 -32328.923,E2 -32328.923} C_VEL
LIN {X 0,Y 5.853,Z 367.032,A -85,B 0,C 180,E1 -32356.021,E2 -32356.021} C_VEL
LIN {X 0,Y 6.287,Z 364.729,A -85,B 0,C 180,E1 -32362.879,E2 -32362.879} C_VEL
LIN {X 0,Y 4.973,Z 375.601,A -85,B 0,C 180,E1 -32398.699,E2 -32398.699} C_VEL
LIN {X 0,Y 3.398,Z 388.918,A -85,B 0,C 180,E1 -32430.86,E2 -32430.86} C_VEL
LIN {X 0,Y 3.652,Z 411.955,A -85,B 0,C 180,E1 -32527.171,E2 -32527.171} C_VEL
LIN {X 0,Y 3.569,Z 411.899,A -85,B 0,C 180,E1 -32532.063,E2 -32532.063} C_VEL
LIN {X 0,Y 3.213,Z 382.363,A -85,B 0,C 180,E1 -32688.502,E2 -32688.502} C_VEL
LIN {X 0,Y 3.233,Z 382.221,A -85,B 0,C 180,E1 -32688.923,E2 -32688.923} C_VEL
LIN {X 0,Y 6.514,Z 382.643,A -85,B 0,C 180,E1 -32716.768,E2 -32716.768} C_VEL
LIN {X 0,Y 6.514,Z 600,A -85,B 0,C 180,E1 -32716.768,E2 -32716.768} C_VEL
LIN {X 0,Y 6.514,Z 600,A -85,B 0,C 180,E1 -32716.768,E2 -32716.768}

QRS_NEXT_CUT()

QRS_NEXT()
QRS_HOME()

END
